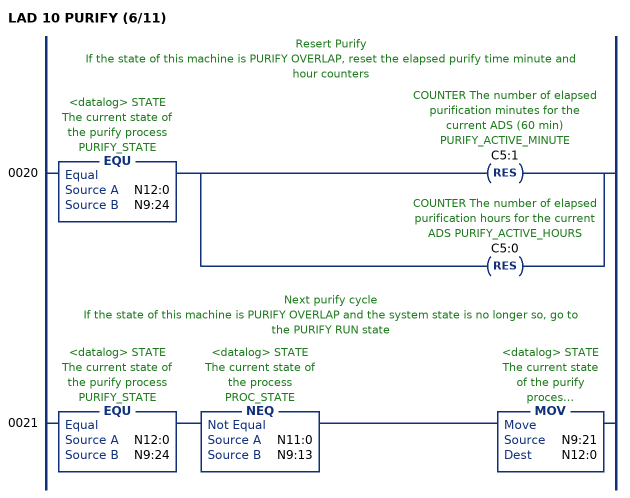
% Rung: 20 %
% Resert Purify
% If the state of this machine is PURIFY OVERLAP, reset the elapsed purify time minute and hour counters %
SOR EQU N12:0 N9:24 BST RES C5:1 NXB RES C5:0 BND EOR
%   N12:0  PURIFY_STATE  "<datalog> STATE The current state of the purify process" %
%   N9:24  PURIFY_OVERLAP  "STATE Puriify Overlap" %
%   C5:1  PURIFY_ACTIVE_MINUTE  "COUNTER The number of elapsed purification minutes for the current ADS (60 min)" %
%   C5:0  PURIFY_ACTIVE_HOURS  "COUNTER The number of elapsed purification hours for the current ADS" %
% Rung: 21 %
% Next purify cycle
% If the state of this machine is PURIFY OVERLAP and the system state is no longer so, go to the PURIFY RUN state %
SOR EQU N12:0 N9:24 NEQ N11:0 N9:13 MOV N9:21 N12:0 EOR
%   N12:0  PURIFY_STATE  "<datalog> STATE The current state of the purify process" %
%   N9:24  PURIFY_OVERLAP  "STATE Puriify Overlap" %
%   N11:0  PROC_STATE  "<datalog> STATE The current state of the process" %
%   N9:13  PROC_OVERLAP  "STATE Process Purify Overlap" %
%   N9:21  PURIFY_RUN  "STATE Purify running" %

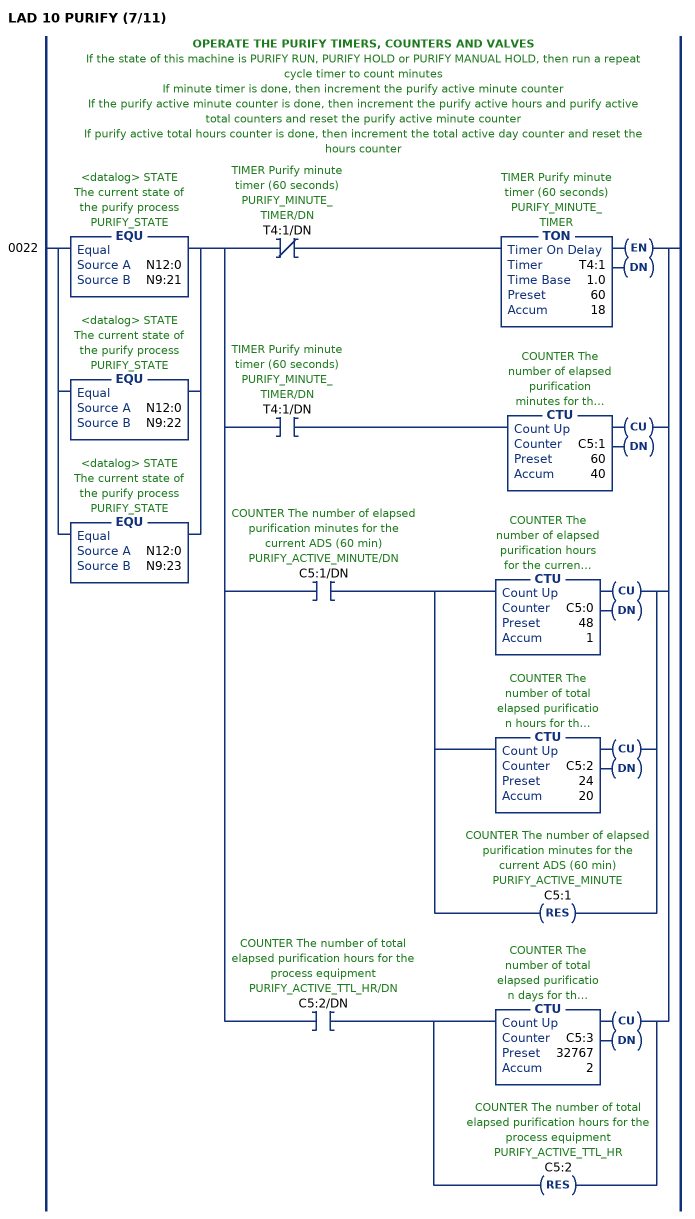
% Rung: 22 %
% TITLE: OPERATE THE PURIFY TIMERS, COUNTERS AND VALVES %
% If the state of this machine is PURIFY RUN, PURIFY HOLD or PURIFY MANUAL HOLD, then run a repeat cycle timer to count minutes
% If minute timer is done, then increment the purify active minute counter
% If the purify active minute counter is done, then increment the purify active hours and purify active total counters and reset the purify active minute counter
% If purify active total hours counter is done, then increment the total active day counter and reset the hours counter %
SOR BST EQU N12:0 N9:21 NXB EQU N12:0 N9:22 NXB EQU N12:0 N9:23 BND BST XIO T4:1/DN TON T4:1 1.0 60 18 NXB XIC T4:1/DN CTU C5:1 60 40 NXB XIC C5:1/DN BST CTU C5:0 48 1 NXB CTU C5:2 24 20 NXB RES C5:1 BND NXB XIC C5:2/DN BST CTU C5:3 32767 2 NXB RES C5:2 BND BND EOR
%   N12:0  PURIFY_STATE  "<datalog> STATE The current state of the purify process" %
%   N9:21  PURIFY_RUN  "STATE Purify running" %
%   N9:22  PURIFY_HOLD  "STATE Purify Hold" %
%   N9:23  PURIFY_MANUAL_HOLD  "STATE Purify Manual Hold" %
%   T4:1  PURIFY_MINUTE_TIMER  "TIMER Purify minute timer (60 seconds)" %
%   C5:1  PURIFY_ACTIVE_MINUTE  "COUNTER The number of elapsed purification minutes for the current ADS (60 min)" %
%   C5:0  PURIFY_ACTIVE_HOURS  "COUNTER The number of elapsed purification hours for the current ADS" %
%   C5:2  PURIFY_ACTIVE_TTL_HR  "COUNTER The number of total elapsed purification hours for the process equipment" %
%   C5:3  PURIFY_ACTIVE_TTL_DY  "COUNTER The number of total elapsed purification days for the process equipment" %

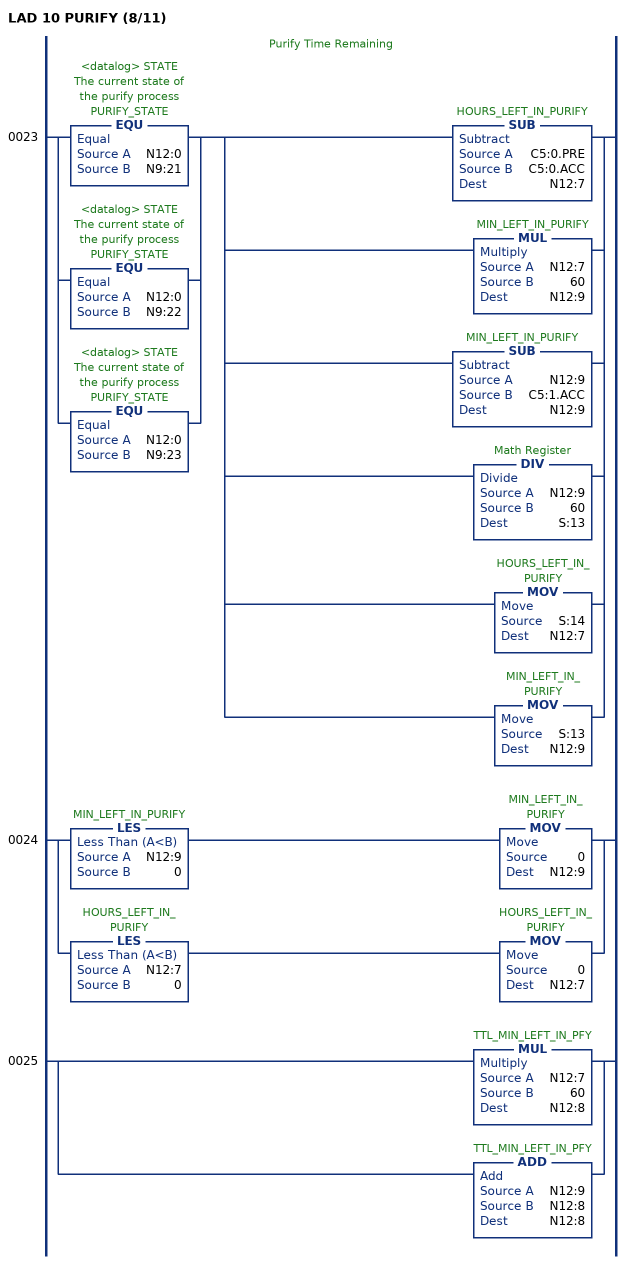
% Rung: 23 %
% Purify Time Remaining %
SOR BST EQU N12:0 N9:21 NXB EQU N12:0 N9:22 NXB EQU N12:0 N9:23 BND BST SUB C5:0.PRE C5:0.ACC N12:7 NXB MUL N12:7 60 N12:9 NXB SUB N12:9 C5:1.ACC N12:9 NXB DIV N12:9 60 S:13 NXB MOV S:14 N12:7 NXB MOV S:13 N12:9 BND EOR
%   N12:0  PURIFY_STATE  "<datalog> STATE The current state of the purify process" %
%   N9:21  PURIFY_RUN  "STATE Purify running" %
%   N9:22  PURIFY_HOLD  "STATE Purify Hold" %
%   N9:23  PURIFY_MANUAL_HOLD  "STATE Purify Manual Hold" %
%   C5:0  PURIFY_ACTIVE_HOURS  "COUNTER The number of elapsed purification hours for the current ADS" %
%   N12:7  HOURS_LEFT_IN_PURIFY %
%   N12:9  MIN_LEFT_IN_PURIFY %
%   C5:1  PURIFY_ACTIVE_MINUTE  "COUNTER The number of elapsed purification minutes for the current ADS (60 min)" %
%   S:13  "Math Register" %
%   S:14  "Math Register" %
% Rung: 24 %
SOR BST LES N12:9 0 MOV 0 N12:9 NXB LES N12:7 0 MOV 0 N12:7 BND EOR
%   N12:9  MIN_LEFT_IN_PURIFY %
%   N12:7  HOURS_LEFT_IN_PURIFY %
% Rung: 25 %
SOR BST MUL N12:7 60 N12:8 NXB ADD N12:9 N12:8 N12:8 BND EOR
%   N12:7  HOURS_LEFT_IN_PURIFY %
%   N12:8  TTL_MIN_LEFT_IN_PFY %
%   N12:9  MIN_LEFT_IN_PURIFY %

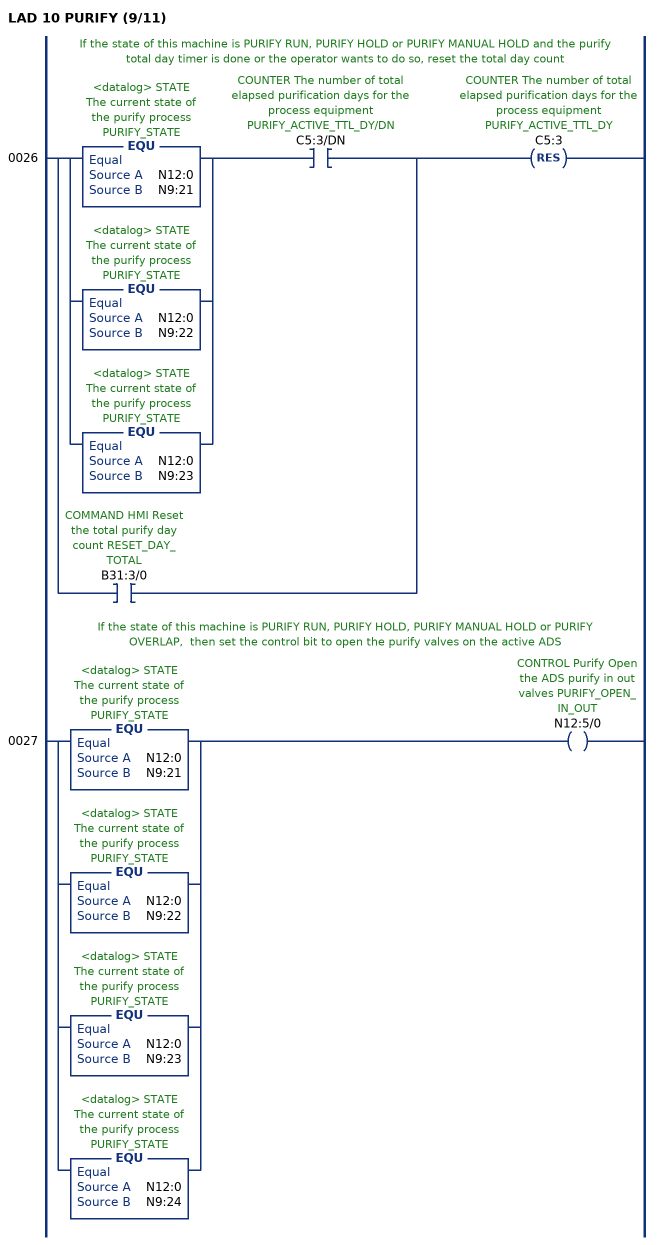
% Rung: 26 %
% If the state of this machine is PURIFY RUN, PURIFY HOLD or PURIFY MANUAL HOLD and the purify total day timer is done or the operator wants to do so, reset the total day count %
SOR BST BST EQU N12:0 N9:21 NXB EQU N12:0 N9:22 NXB EQU N12:0 N9:23 BND XIC C5:3/DN NXB XIC B31:3/0 BND RES C5:3 EOR
%   N12:0  PURIFY_STATE  "<datalog> STATE The current state of the purify process" %
%   N9:21  PURIFY_RUN  "STATE Purify running" %
%   N9:22  PURIFY_HOLD  "STATE Purify Hold" %
%   N9:23  PURIFY_MANUAL_HOLD  "STATE Purify Manual Hold" %
%   C5:3  PURIFY_ACTIVE_TTL_DY  "COUNTER The number of total elapsed purification days for the process equipment" %
%   B31:3/0  RESET_DAY_TOTAL  "COMMAND HMI Reset the total purify day count" %
% Rung: 27 %
% If the state of this machine is PURIFY RUN, PURIFY HOLD, PURIFY MANUAL HOLD or PURIFY OVERLAP,  then set the control bit to open the purify valves on the active ADS %
SOR BST EQU N12:0 N9:21 NXB EQU N12:0 N9:22 NXB EQU N12:0 N9:23 NXB EQU N12:0 N9:24 BND OTE N12:5/0 EOR
%   N12:0  PURIFY_STATE  "<datalog> STATE The current state of the purify process" %
%   N9:21  PURIFY_RUN  "STATE Purify running" %
%   N9:22  PURIFY_HOLD  "STATE Purify Hold" %
%   N9:23  PURIFY_MANUAL_HOLD  "STATE Purify Manual Hold" %
%   N9:24  PURIFY_OVERLAP  "STATE Puriify Overlap" %
%   N12:5/0  PURIFY_OPEN_IN_OUT  "CONTROL Purify Open the ADS purify in out valves" %

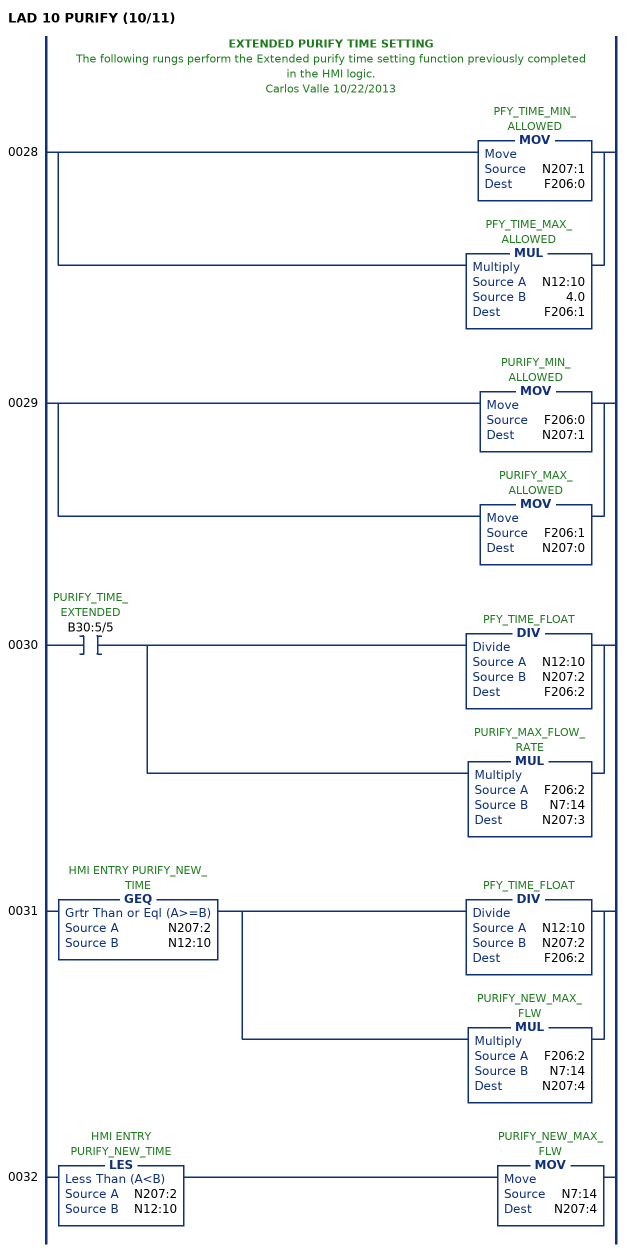
% Rung: 28 %
% TITLE: EXTENDED PURIFY TIME SETTING %
% The following rungs perform the Extended purify time setting function previously completed in the HMI logic.
% Carlos Valle 10/22/2013 %
SOR BST MOV N207:1 F206:0 NXB MUL N12:10 4.0 F206:1 BND EOR
%   N207:1  PURIFY_MIN_ALLOWED %
%   F206:0  PFY_TIME_MIN_ALLOWED %
%   N12:10  DEFAULT_PURIFY_TIME  "CONFIG The percent output requested by the operator (percent)" %
%   F206:1  PFY_TIME_MAX_ALLOWED %
% Rung: 29 %
SOR BST MOV F206:0 N207:1 NXB MOV F206:1 N207:0 BND EOR
%   F206:0  PFY_TIME_MIN_ALLOWED %
%   N207:1  PURIFY_MIN_ALLOWED %
%   F206:1  PFY_TIME_MAX_ALLOWED %
%   N207:0  PURIFY_MAX_ALLOWED %
% Rung: 30 %
SOR XIC B30:5/5 BST DIV N12:10 N207:2 F206:2 NXB MUL F206:2 N7:14 N207:3 BND EOR
%   B30:5/5  PURIFY_TIME_EXTENDED %
%   N12:10  DEFAULT_PURIFY_TIME  "CONFIG The percent output requested by the operator (percent)" %
%   N207:2  PURIFY_NEW_TIME  "HMI ENTRY" %
%   F206:2  PFY_TIME_FLOAT %
%   N7:14  PURIFIER_SIZE %
%   N207:3  PURIFY_MAX_FLOW_RATE %
% Rung: 31 %
SOR GEQ N207:2 N12:10 BST DIV N12:10 N207:2 F206:2 NXB MUL F206:2 N7:14 N207:4 BND EOR
%   N207:2  PURIFY_NEW_TIME  "HMI ENTRY" %
%   N12:10  DEFAULT_PURIFY_TIME  "CONFIG The percent output requested by the operator (percent)" %
%   F206:2  PFY_TIME_FLOAT %
%   N7:14  PURIFIER_SIZE %
%   N207:4  PURIFY_NEW_MAX_FLW %
% Rung: 32 %
SOR LES N207:2 N12:10 MOV N7:14 N207:4 EOR
%   N207:2  PURIFY_NEW_TIME  "HMI ENTRY" %
%   N12:10  DEFAULT_PURIFY_TIME  "CONFIG The percent output requested by the operator (percent)" %
%   N7:14  PURIFIER_SIZE %
%   N207:4  PURIFY_NEW_MAX_FLW %

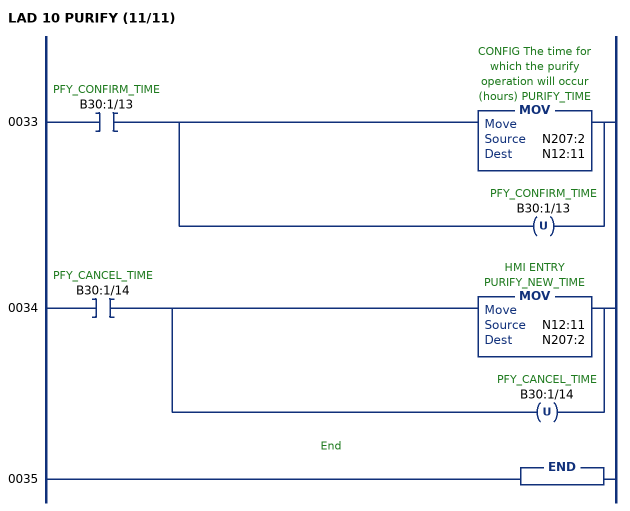
% Rung: 33 %
SOR XIC B30:1/13 BST MOV N207:2 N12:11 NXB OTU B30:1/13 BND EOR
%   B30:1/13  PFY_CONFIRM_TIME %
%   N207:2  PURIFY_NEW_TIME  "HMI ENTRY" %
%   N12:11  PURIFY_TIME  "CONFIG The time for which the purify operation will occur (hours)" %
% Rung: 34 %
SOR XIC B30:1/14 BST MOV N12:11 N207:2 NXB OTU B30:1/14 BND EOR
%   B30:1/14  PFY_CANCEL_TIME %
%   N12:11  PURIFY_TIME  "CONFIG The time for which the purify operation will occur (hours)" %
%   N207:2  PURIFY_NEW_TIME  "HMI ENTRY" %
% Rung: 35 %
% End %
SOR END EOR

LADDER 11 "REGEN"    % Operates the regen control %
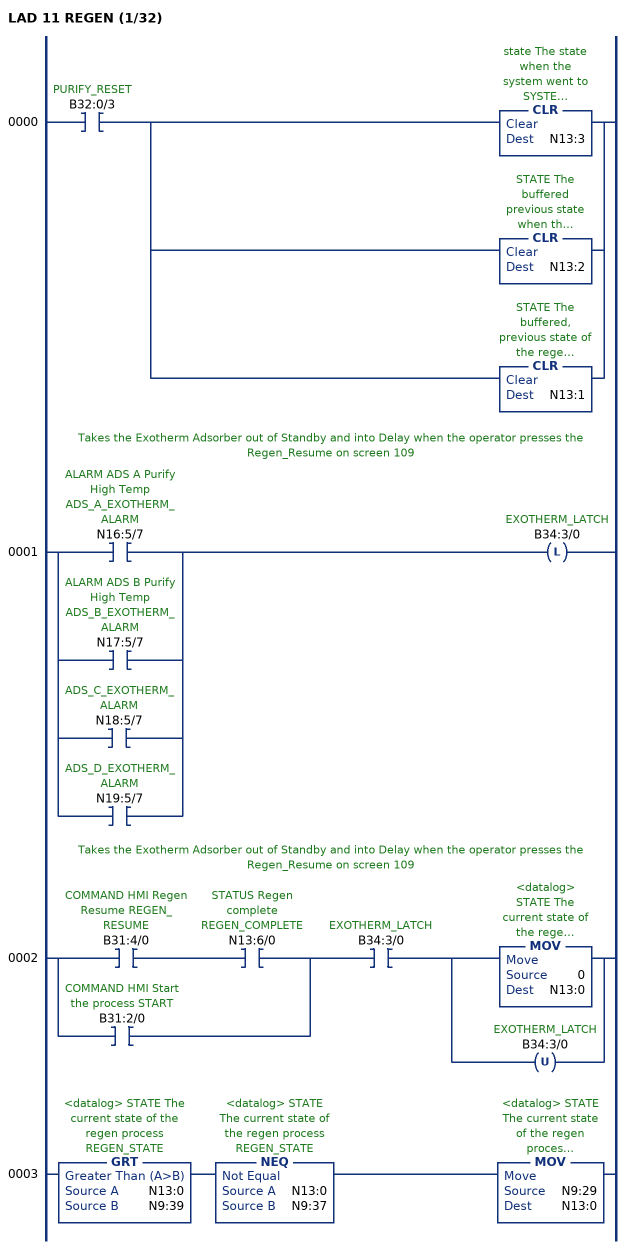
% Rung: 0 %
SOR XIC B32:0/3 BST CLR N13:3 NXB CLR N13:2 NXB CLR N13:1 BND EOR
%   B32:0/3  PURIFY_RESET %
%   N13:3  REGEN_STANDBY_BUFFER  "state The state when the system went to SYSTEM STANDBY" %
%   N13:2  REGEN_ALARM_BUFFER  "STATE The buffered previous state when the system alarm occured" %
%   N13:1  REGEN_BUFFER  "STATE The buffered, previous state of the regen process" %
% Rung: 1 %
% Takes the Exotherm Adsorber out of Standby and into Delay when the operator presses the Regen_Resume on screen 109 %
SOR BST XIC N16:5/7 NXB XIC N17:5/7 NXB XIC N18:5/7 NXB XIC N19:5/7 BND OTL B34:3/0 EOR
%   N16:5/7  ADS_A_EXOTHERM_ALARM  "ALARM ADS A Purify High Temp" %
%   N17:5/7  ADS_B_EXOTHERM_ALARM  "ALARM ADS B Purify High Temp" %
%   N18:5/7  ADS_C_EXOTHERM_ALARM %
%   N19:5/7  ADS_D_EXOTHERM_ALARM %
%   B34:3/0  EXOTHERM_LATCH %
% Rung: 2 %
% Takes the Exotherm Adsorber out of Standby and into Delay when the operator presses the Regen_Resume on screen 109 %
SOR BST XIC B31:4/0 XIC N13:6/0 NXB XIC B31:2/0 BND XIC B34:3/0 BST MOV 0 N13:0 NXB OTU B34:3/0 BND EOR
%   B31:4/0  REGEN_RESUME  "COMMAND HMI Regen Resume" %
%   N13:6/0  REGEN_COMPLETE  "STATUS Regen complete" %
%   B31:2/0  START  "COMMAND HMI Start the process" %
%   B34:3/0  EXOTHERM_LATCH %
%   N13:0  REGEN_STATE  "<datalog> STATE The current state of the regen process" %
% Rung: 3 %
SOR GRT N13:0 N9:39 NEQ N13:0 N9:37 MOV N9:29 N13:0 EOR
%   N13:0  REGEN_STATE  "<datalog> STATE The current state of the regen process" %
%   N9:39  REGEN_EQUALIZE  "STATE Regen Equalize" %
%   N9:37  REGEN_ALARM  "STATE Regen Alarm" %
%   N9:29  REGEN_IDLE  "STATE Regen Idle" %

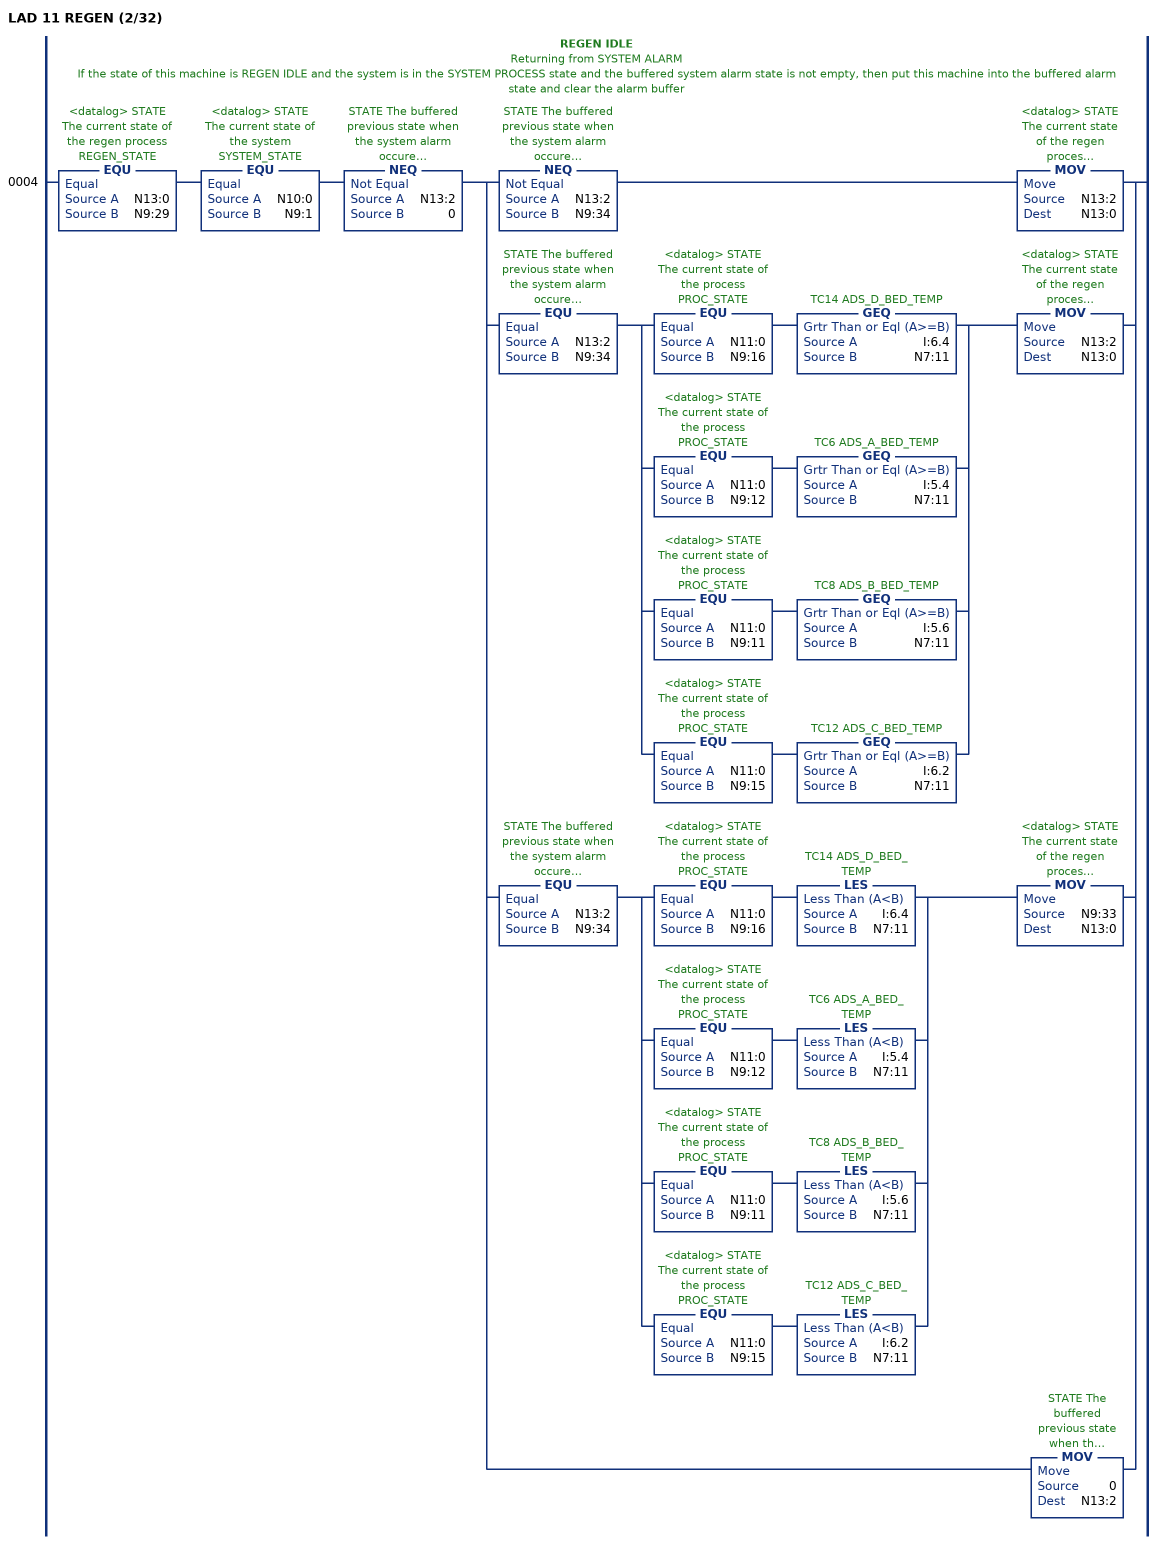
% Rung: 4 %
% TITLE: REGEN IDLE %
% Returning from SYSTEM ALARM
% If the state of this machine is REGEN IDLE and the system is in the SYSTEM PROCESS state and the buffered system alarm state is not empty, then put this machine into the buffered alarm state and clear the alarm buffer %
SOR EQU N13:0 N9:29 EQU N10:0 N9:1 NEQ N13:2 0 BST NEQ N13:2 N9:34 MOV N13:2 N13:0 NXB EQU N13:2 N9:34 BST EQU N11:0 N9:16 GEQ I:6.4 N7:11 NXB EQU N11:0 N9:12 GEQ I:5.4 N7:11 NXB EQU N11:0 N9:11 GEQ I:5.6 N7:11 NXB EQU N11:0 N9:15 GEQ I:6.2 N7:11 BND MOV N13:2 N13:0 NXB EQU N13:2 N9:34 BST EQU N11:0 N9:16 LES I:6.4 N7:11 NXB EQU N11:0 N9:12 LES I:5.4 N7:11 NXB EQU N11:0 N9:11 LES I:5.6 N7:11 NXB EQU N11:0 N9:15 LES I:6.2 N7:11 BND MOV N9:33 N13:0 NXB MOV 0 N13:2 BND EOR
%   N13:0  REGEN_STATE  "<datalog> STATE The current state of the regen process" %
%   N9:29  REGEN_IDLE  "STATE Regen Idle" %
%   N10:0  SYSTEM_STATE  "<datalog> STATE The current state of the system" %
%   N9:1  SYSTEM_PROCESS  "STATE System Process" %
%   N13:2  REGEN_ALARM_BUFFER  "STATE The buffered previous state when the system alarm occured" %
%   N9:34  REGEN_H2_REDUCTION  "STATE Regen Running" %
%   N11:0  PROC_STATE  "<datalog> STATE The current state of the process" %
%   N9:16  PROC_REGEN_D  "STATE Process Regen D" %
%   I:6.4  ADS_D_BED_TEMP  "TC14" %
%   N7:11  ADS_BED_TEMP_HIGH  "CONFIG The temp at which the regen process may continue" %
%   N9:12  PROC_REGEN_A  "STATE Process Regen A" %
%   I:5.4  ADS_A_BED_TEMP  "TC6" %
%   N9:11  PROC_REGEN_B  "STATE Process Regen B" %
%   I:5.6  ADS_B_BED_TEMP  "TC8" %
%   N9:15  PROC_REGEN_C  "STATE Process Regen C" %
%   I:6.2  ADS_C_BED_TEMP  "TC12" %
%   N9:33  REGEN_HEAT_BED  "STATE Regen Heat wall" %

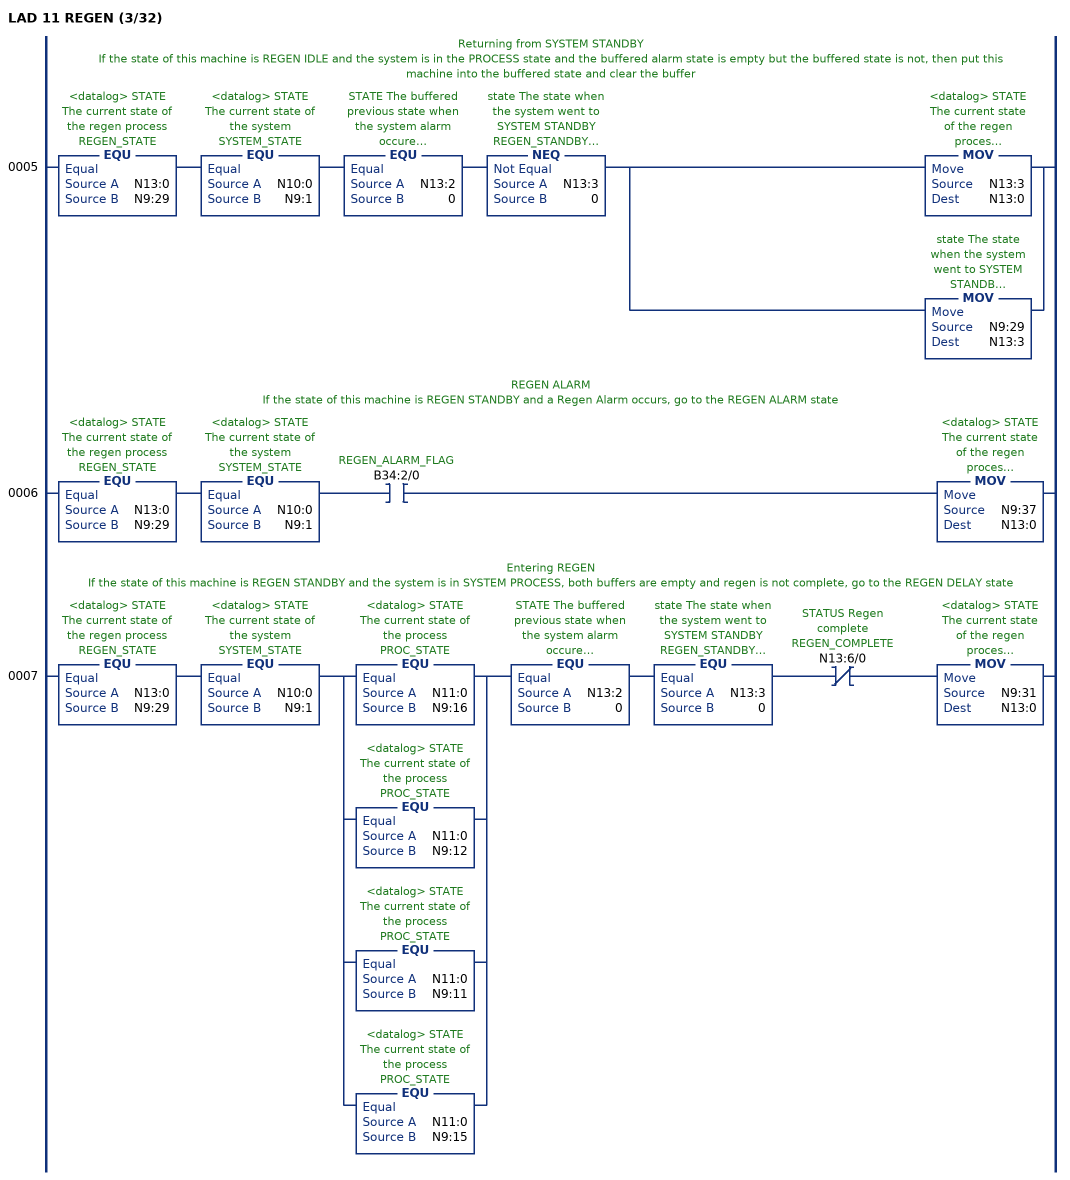
% Rung: 5 %
% Returning from SYSTEM STANDBY
% If the state of this machine is REGEN IDLE and the system is in the PROCESS state and the buffered alarm state is empty but the buffered state is not, then put this machine into the buffered state and clear the buffer %
SOR EQU N13:0 N9:29 EQU N10:0 N9:1 EQU N13:2 0 NEQ N13:3 0 BST MOV N13:3 N13:0 NXB MOV N9:29 N13:3 BND EOR
%   N13:0  REGEN_STATE  "<datalog> STATE The current state of the regen process" %
%   N9:29  REGEN_IDLE  "STATE Regen Idle" %
%   N10:0  SYSTEM_STATE  "<datalog> STATE The current state of the system" %
%   N9:1  SYSTEM_PROCESS  "STATE System Process" %
%   N13:2  REGEN_ALARM_BUFFER  "STATE The buffered previous state when the system alarm occured" %
%   N13:3  REGEN_STANDBY_BUFFER  "state The state when the system went to SYSTEM STANDBY" %
% Rung: 6 %
% REGEN ALARM
% If the state of this machine is REGEN STANDBY and a Regen Alarm occurs, go to the REGEN ALARM state %
SOR EQU N13:0 N9:29 EQU N10:0 N9:1 XIC B34:2/0 MOV N9:37 N13:0 EOR
%   N13:0  REGEN_STATE  "<datalog> STATE The current state of the regen process" %
%   N9:29  REGEN_IDLE  "STATE Regen Idle" %
%   N10:0  SYSTEM_STATE  "<datalog> STATE The current state of the system" %
%   N9:1  SYSTEM_PROCESS  "STATE System Process" %
%   B34:2/0  REGEN_ALARM_FLAG %
%   N9:37  REGEN_ALARM  "STATE Regen Alarm" %
% Rung: 7 %
% Entering REGEN
% If the state of this machine is REGEN STANDBY and the system is in SYSTEM PROCESS, both buffers are empty and regen is not complete, go to the REGEN DELAY state %
SOR EQU N13:0 N9:29 EQU N10:0 N9:1 BST EQU N11:0 N9:16 NXB EQU N11:0 N9:12 NXB EQU N11:0 N9:11 NXB EQU N11:0 N9:15 BND EQU N13:2 0 EQU N13:3 0 XIO N13:6/0 MOV N9:31 N13:0 EOR
%   N13:0  REGEN_STATE  "<datalog> STATE The current state of the regen process" %
%   N9:29  REGEN_IDLE  "STATE Regen Idle" %
%   N10:0  SYSTEM_STATE  "<datalog> STATE The current state of the system" %
%   N9:1  SYSTEM_PROCESS  "STATE System Process" %
%   N11:0  PROC_STATE  "<datalog> STATE The current state of the process" %
%   N9:16  PROC_REGEN_D  "STATE Process Regen D" %
%   N9:12  PROC_REGEN_A  "STATE Process Regen A" %
%   N9:11  PROC_REGEN_B  "STATE Process Regen B" %
%   N9:15  PROC_REGEN_C  "STATE Process Regen C" %
%   N13:2  REGEN_ALARM_BUFFER  "STATE The buffered previous state when the system alarm occured" %
%   N13:3  REGEN_STANDBY_BUFFER  "state The state when the system went to SYSTEM STANDBY" %
%   N13:6/0  REGEN_COMPLETE  "STATUS Regen complete" %
%   N9:31  REGEN_DELAY  "STATE Regen Delay" %

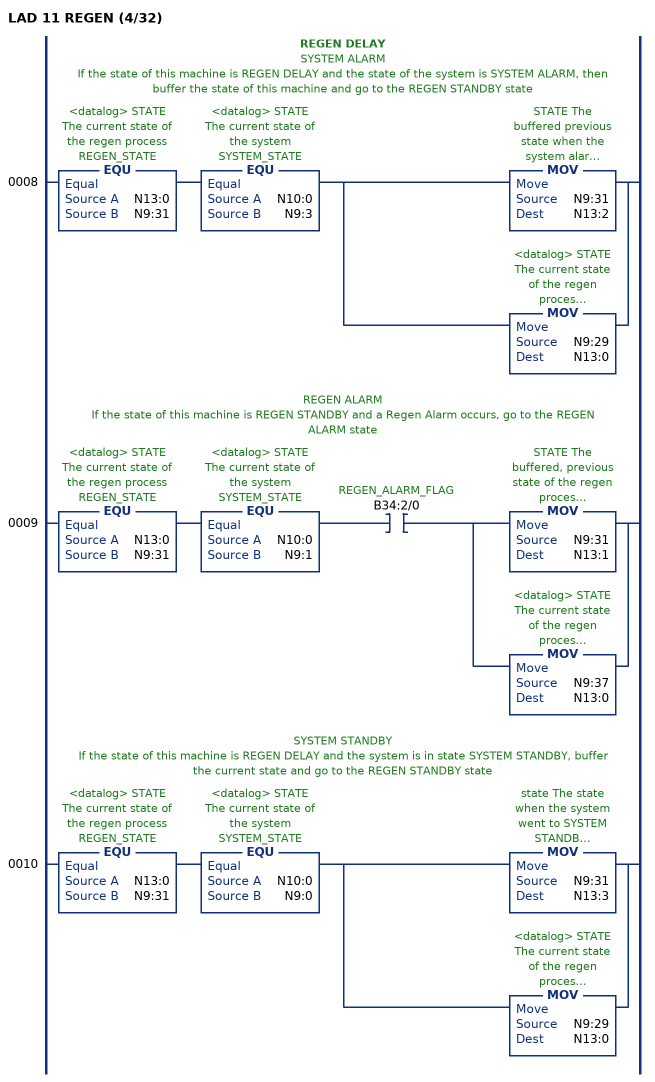
% Rung: 8 %
% TITLE: REGEN DELAY %
% SYSTEM ALARM
% If the state of this machine is REGEN DELAY and the state of the system is SYSTEM ALARM, then buffer the state of this machine and go to the REGEN STANDBY state %
SOR EQU N13:0 N9:31 EQU N10:0 N9:3 BST MOV N9:31 N13:2 NXB MOV N9:29 N13:0 BND EOR
%   N13:0  REGEN_STATE  "<datalog> STATE The current state of the regen process" %
%   N9:31  REGEN_DELAY  "STATE Regen Delay" %
%   N10:0  SYSTEM_STATE  "<datalog> STATE The current state of the system" %
%   N9:3  SYSTEM_ALARM  "STATE System Alarm" %
%   N13:2  REGEN_ALARM_BUFFER  "STATE The buffered previous state when the system alarm occured" %
%   N9:29  REGEN_IDLE  "STATE Regen Idle" %
% Rung: 9 %
% REGEN ALARM
% If the state of this machine is REGEN STANDBY and a Regen Alarm occurs, go to the REGEN ALARM state %
SOR EQU N13:0 N9:31 EQU N10:0 N9:1 XIC B34:2/0 BST MOV N9:31 N13:1 NXB MOV N9:37 N13:0 BND EOR
%   N13:0  REGEN_STATE  "<datalog> STATE The current state of the regen process" %
%   N9:31  REGEN_DELAY  "STATE Regen Delay" %
%   N10:0  SYSTEM_STATE  "<datalog> STATE The current state of the system" %
%   N9:1  SYSTEM_PROCESS  "STATE System Process" %
%   B34:2/0  REGEN_ALARM_FLAG %
%   N13:1  REGEN_BUFFER  "STATE The buffered, previous state of the regen process" %
%   N9:37  REGEN_ALARM  "STATE Regen Alarm" %
% Rung: 10 %
% SYSTEM STANDBY
% If the state of this machine is REGEN DELAY and the system is in state SYSTEM STANDBY, buffer the current state and go to the REGEN STANDBY state %
SOR EQU N13:0 N9:31 EQU N10:0 N9:0 BST MOV N9:31 N13:3 NXB MOV N9:29 N13:0 BND EOR
%   N13:0  REGEN_STATE  "<datalog> STATE The current state of the regen process" %
%   N9:31  REGEN_DELAY  "STATE Regen Delay" %
%   N10:0  SYSTEM_STATE  "<datalog> STATE The current state of the system" %
%   N9:0  SYSTEM_STANDBY  "STATE System Standby" %
%   N13:3  REGEN_STANDBY_BUFFER  "state The state when the system went to SYSTEM STANDBY" %
%   N9:29  REGEN_IDLE  "STATE Regen Idle" %

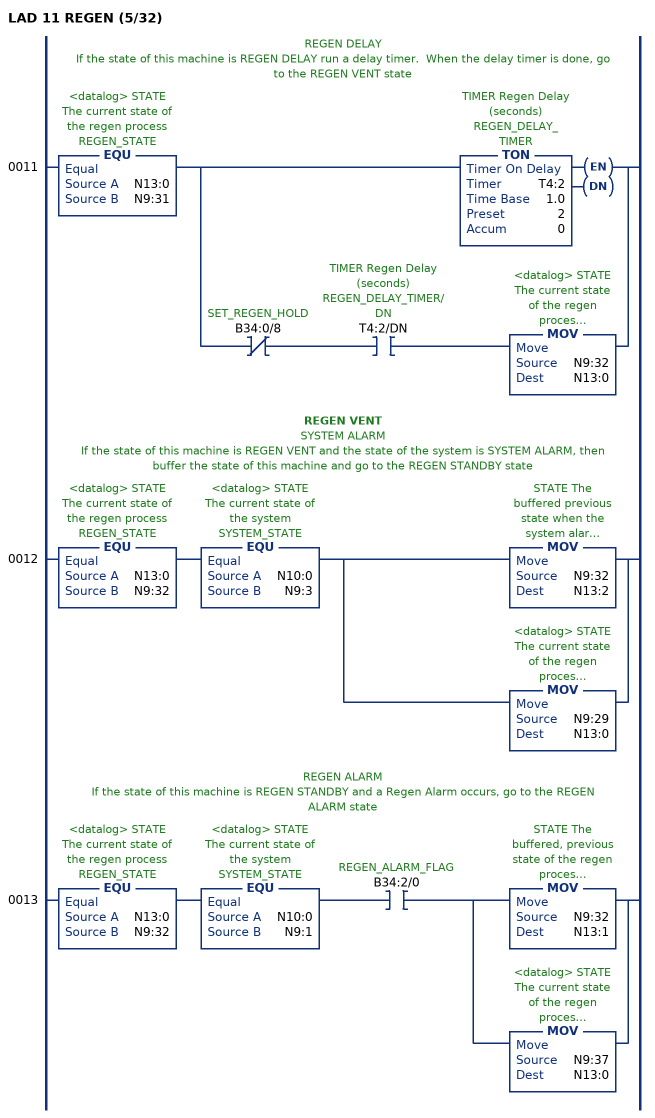
% Rung: 11 %
% REGEN DELAY
% If the state of this machine is REGEN DELAY run a delay timer.  When the delay timer is done, go to the REGEN VENT state %
SOR EQU N13:0 N9:31 BST TON T4:2 1.0 2 0 NXB XIO B34:0/8 XIC T4:2/DN MOV N9:32 N13:0 BND EOR
%   N13:0  REGEN_STATE  "<datalog> STATE The current state of the regen process" %
%   N9:31  REGEN_DELAY  "STATE Regen Delay" %
%   T4:2  REGEN_DELAY_TIMER  "TIMER Regen Delay (seconds)" %
%   B34:0/8  SET_REGEN_HOLD %
%   N9:32  REGEN_VENT  "STATE Regen Vent" %
% Rung: 12 %
% TITLE: REGEN VENT %
% SYSTEM ALARM
% If the state of this machine is REGEN VENT and the state of the system is SYSTEM ALARM, then buffer the state of this machine and go to the REGEN STANDBY state %
SOR EQU N13:0 N9:32 EQU N10:0 N9:3 BST MOV N9:32 N13:2 NXB MOV N9:29 N13:0 BND EOR
%   N13:0  REGEN_STATE  "<datalog> STATE The current state of the regen process" %
%   N9:32  REGEN_VENT  "STATE Regen Vent" %
%   N10:0  SYSTEM_STATE  "<datalog> STATE The current state of the system" %
%   N9:3  SYSTEM_ALARM  "STATE System Alarm" %
%   N13:2  REGEN_ALARM_BUFFER  "STATE The buffered previous state when the system alarm occured" %
%   N9:29  REGEN_IDLE  "STATE Regen Idle" %
% Rung: 13 %
% REGEN ALARM
% If the state of this machine is REGEN STANDBY and a Regen Alarm occurs, go to the REGEN ALARM state %
SOR EQU N13:0 N9:32 EQU N10:0 N9:1 XIC B34:2/0 BST MOV N9:32 N13:1 NXB MOV N9:37 N13:0 BND EOR
%   N13:0  REGEN_STATE  "<datalog> STATE The current state of the regen process" %
%   N9:32  REGEN_VENT  "STATE Regen Vent" %
%   N10:0  SYSTEM_STATE  "<datalog> STATE The current state of the system" %
%   N9:1  SYSTEM_PROCESS  "STATE System Process" %
%   B34:2/0  REGEN_ALARM_FLAG %
%   N13:1  REGEN_BUFFER  "STATE The buffered, previous state of the regen process" %
%   N9:37  REGEN_ALARM  "STATE Regen Alarm" %

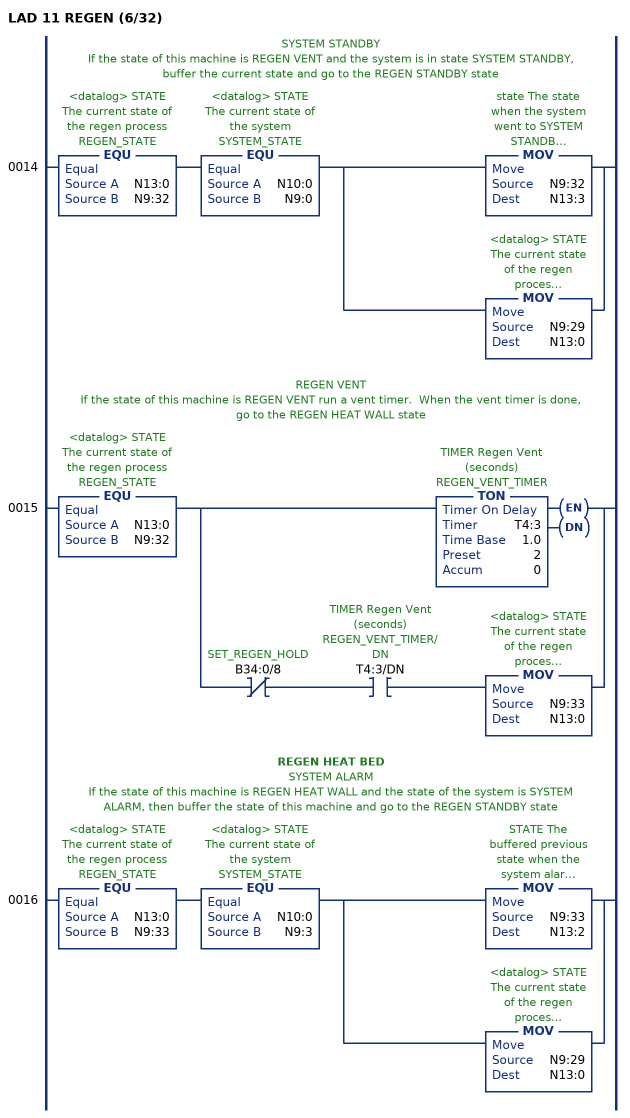
% Rung: 14 %
% SYSTEM STANDBY
% If the state of this machine is REGEN VENT and the system is in state SYSTEM STANDBY, buffer the current state and go to the REGEN STANDBY state %
SOR EQU N13:0 N9:32 EQU N10:0 N9:0 BST MOV N9:32 N13:3 NXB MOV N9:29 N13:0 BND EOR
%   N13:0  REGEN_STATE  "<datalog> STATE The current state of the regen process" %
%   N9:32  REGEN_VENT  "STATE Regen Vent" %
%   N10:0  SYSTEM_STATE  "<datalog> STATE The current state of the system" %
%   N9:0  SYSTEM_STANDBY  "STATE System Standby" %
%   N13:3  REGEN_STANDBY_BUFFER  "state The state when the system went to SYSTEM STANDBY" %
%   N9:29  REGEN_IDLE  "STATE Regen Idle" %
% Rung: 15 %
% REGEN VENT
% If the state of this machine is REGEN VENT run a vent timer.  When the vent timer is done, go to the REGEN HEAT WALL state %
SOR EQU N13:0 N9:32 BST TON T4:3 1.0 2 0 NXB XIO B34:0/8 XIC T4:3/DN MOV N9:33 N13:0 BND EOR
%   N13:0  REGEN_STATE  "<datalog> STATE The current state of the regen process" %
%   N9:32  REGEN_VENT  "STATE Regen Vent" %
%   T4:3  REGEN_VENT_TIMER  "TIMER Regen Vent (seconds)" %
%   B34:0/8  SET_REGEN_HOLD %
%   N9:33  REGEN_HEAT_BED  "STATE Regen Heat wall" %
% Rung: 16 %
% TITLE: REGEN HEAT BED %
% SYSTEM ALARM
% If the state of this machine is REGEN HEAT WALL and the state of the system is SYSTEM ALARM, then buffer the state of this machine and go to the REGEN STANDBY state %
SOR EQU N13:0 N9:33 EQU N10:0 N9:3 BST MOV N9:33 N13:2 NXB MOV N9:29 N13:0 BND EOR
%   N13:0  REGEN_STATE  "<datalog> STATE The current state of the regen process" %
%   N9:33  REGEN_HEAT_BED  "STATE Regen Heat wall" %
%   N10:0  SYSTEM_STATE  "<datalog> STATE The current state of the system" %
%   N9:3  SYSTEM_ALARM  "STATE System Alarm" %
%   N13:2  REGEN_ALARM_BUFFER  "STATE The buffered previous state when the system alarm occured" %
%   N9:29  REGEN_IDLE  "STATE Regen Idle" %

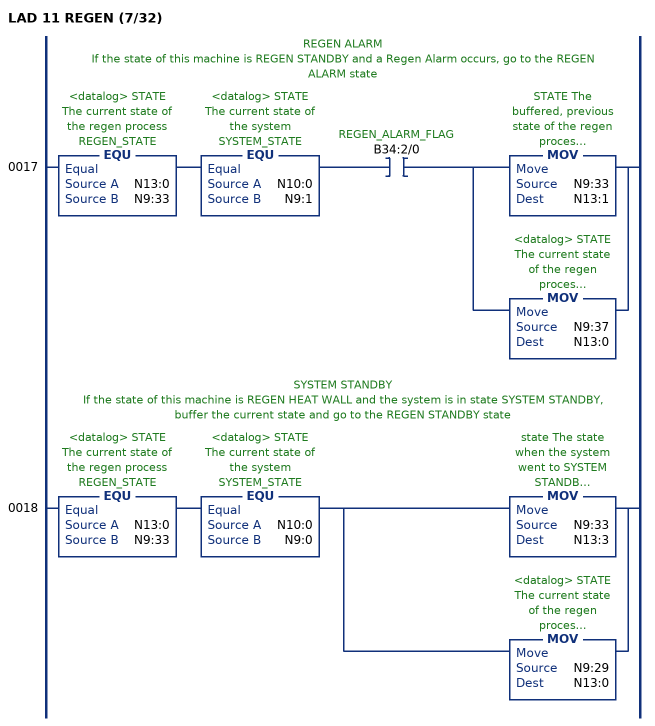
% Rung: 17 %
% REGEN ALARM
% If the state of this machine is REGEN STANDBY and a Regen Alarm occurs, go to the REGEN ALARM state %
SOR EQU N13:0 N9:33 EQU N10:0 N9:1 XIC B34:2/0 BST MOV N9:33 N13:1 NXB MOV N9:37 N13:0 BND EOR
%   N13:0  REGEN_STATE  "<datalog> STATE The current state of the regen process" %
%   N9:33  REGEN_HEAT_BED  "STATE Regen Heat wall" %
%   N10:0  SYSTEM_STATE  "<datalog> STATE The current state of the system" %
%   N9:1  SYSTEM_PROCESS  "STATE System Process" %
%   B34:2/0  REGEN_ALARM_FLAG %
%   N13:1  REGEN_BUFFER  "STATE The buffered, previous state of the regen process" %
%   N9:37  REGEN_ALARM  "STATE Regen Alarm" %
% Rung: 18 %
% SYSTEM STANDBY
% If the state of this machine is REGEN HEAT WALL and the system is in state SYSTEM STANDBY, buffer the current state and go to the REGEN STANDBY state %
SOR EQU N13:0 N9:33 EQU N10:0 N9:0 BST MOV N9:33 N13:3 NXB MOV N9:29 N13:0 BND EOR
%   N13:0  REGEN_STATE  "<datalog> STATE The current state of the regen process" %
%   N9:33  REGEN_HEAT_BED  "STATE Regen Heat wall" %
%   N10:0  SYSTEM_STATE  "<datalog> STATE The current state of the system" %
%   N9:0  SYSTEM_STANDBY  "STATE System Standby" %
%   N13:3  REGEN_STANDBY_BUFFER  "state The state when the system went to SYSTEM STANDBY" %
%   N9:29  REGEN_IDLE  "STATE Regen Idle" %

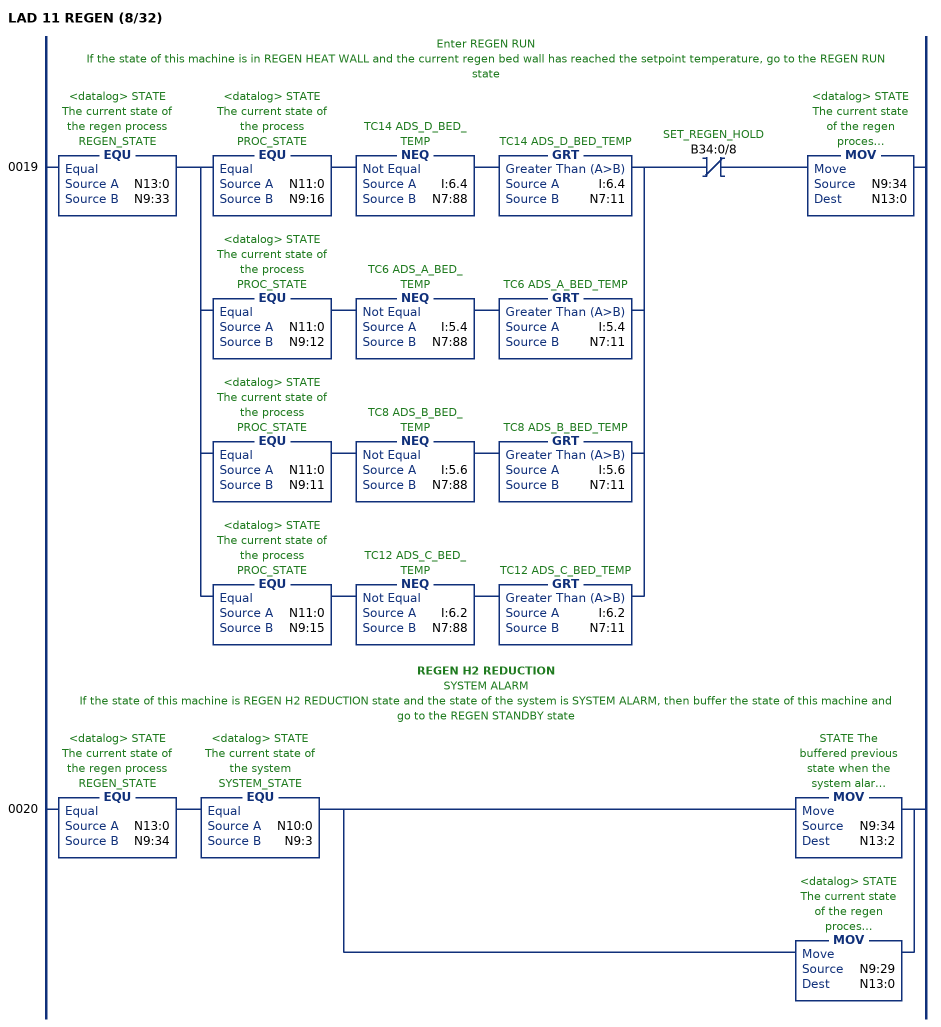
% Rung: 19 %
% Enter REGEN RUN
% If the state of this machine is in REGEN HEAT WALL and the current regen bed wall has reached the setpoint temperature, go to the REGEN RUN state %
SOR EQU N13:0 N9:33 BST EQU N11:0 N9:16 NEQ I:6.4 N7:88 GRT I:6.4 N7:11 NXB EQU N11:0 N9:12 NEQ I:5.4 N7:88 GRT I:5.4 N7:11 NXB EQU N11:0 N9:11 NEQ I:5.6 N7:88 GRT I:5.6 N7:11 NXB EQU N11:0 N9:15 NEQ I:6.2 N7:88 GRT I:6.2 N7:11 BND XIO B34:0/8 MOV N9:34 N13:0 EOR
%   N13:0  REGEN_STATE  "<datalog> STATE The current state of the regen process" %
%   N9:33  REGEN_HEAT_BED  "STATE Regen Heat wall" %
%   N11:0  PROC_STATE  "<datalog> STATE The current state of the process" %
%   N9:16  PROC_REGEN_D  "STATE Process Regen D" %
%   I:6.4  ADS_D_BED_TEMP  "TC14" %
%   N7:88  TC_OPEN_SP  "CONFIG TC Open Setpoint" %
%   N7:11  ADS_BED_TEMP_HIGH  "CONFIG The temp at which the regen process may continue" %
%   N9:12  PROC_REGEN_A  "STATE Process Regen A" %
%   I:5.4  ADS_A_BED_TEMP  "TC6" %
%   N9:11  PROC_REGEN_B  "STATE Process Regen B" %
%   I:5.6  ADS_B_BED_TEMP  "TC8" %
%   N9:15  PROC_REGEN_C  "STATE Process Regen C" %
%   I:6.2  ADS_C_BED_TEMP  "TC12" %
%   B34:0/8  SET_REGEN_HOLD %
%   N9:34  REGEN_H2_REDUCTION  "STATE Regen Running" %
% Rung: 20 %
% TITLE: REGEN H2 REDUCTION %
% SYSTEM ALARM
% If the state of this machine is REGEN H2 REDUCTION state and the state of the system is SYSTEM ALARM, then buffer the state of this machine and go to the REGEN STANDBY state %
SOR EQU N13:0 N9:34 EQU N10:0 N9:3 BST MOV N9:34 N13:2 NXB MOV N9:29 N13:0 BND EOR
%   N13:0  REGEN_STATE  "<datalog> STATE The current state of the regen process" %
%   N9:34  REGEN_H2_REDUCTION  "STATE Regen Running" %
%   N10:0  SYSTEM_STATE  "<datalog> STATE The current state of the system" %
%   N9:3  SYSTEM_ALARM  "STATE System Alarm" %
%   N13:2  REGEN_ALARM_BUFFER  "STATE The buffered previous state when the system alarm occured" %
%   N9:29  REGEN_IDLE  "STATE Regen Idle" %

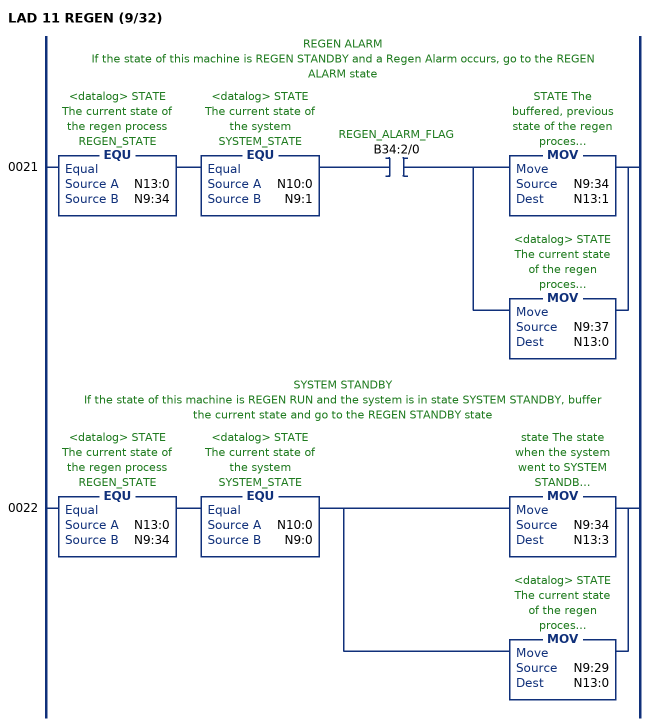
% Rung: 21 %
% REGEN ALARM
% If the state of this machine is REGEN STANDBY and a Regen Alarm occurs, go to the REGEN ALARM state %
SOR EQU N13:0 N9:34 EQU N10:0 N9:1 XIC B34:2/0 BST MOV N9:34 N13:1 NXB MOV N9:37 N13:0 BND EOR
%   N13:0  REGEN_STATE  "<datalog> STATE The current state of the regen process" %
%   N9:34  REGEN_H2_REDUCTION  "STATE Regen Running" %
%   N10:0  SYSTEM_STATE  "<datalog> STATE The current state of the system" %
%   N9:1  SYSTEM_PROCESS  "STATE System Process" %
%   B34:2/0  REGEN_ALARM_FLAG %
%   N13:1  REGEN_BUFFER  "STATE The buffered, previous state of the regen process" %
%   N9:37  REGEN_ALARM  "STATE Regen Alarm" %
% Rung: 22 %
% SYSTEM STANDBY
% If the state of this machine is REGEN RUN and the system is in state SYSTEM STANDBY, buffer the current state and go to the REGEN STANDBY state %
SOR EQU N13:0 N9:34 EQU N10:0 N9:0 BST MOV N9:34 N13:3 NXB MOV N9:29 N13:0 BND EOR
%   N13:0  REGEN_STATE  "<datalog> STATE The current state of the regen process" %
%   N9:34  REGEN_H2_REDUCTION  "STATE Regen Running" %
%   N10:0  SYSTEM_STATE  "<datalog> STATE The current state of the system" %
%   N9:0  SYSTEM_STANDBY  "STATE System Standby" %
%   N13:3  REGEN_STANDBY_BUFFER  "state The state when the system went to SYSTEM STANDBY" %
%   N9:29  REGEN_IDLE  "STATE Regen Idle" %

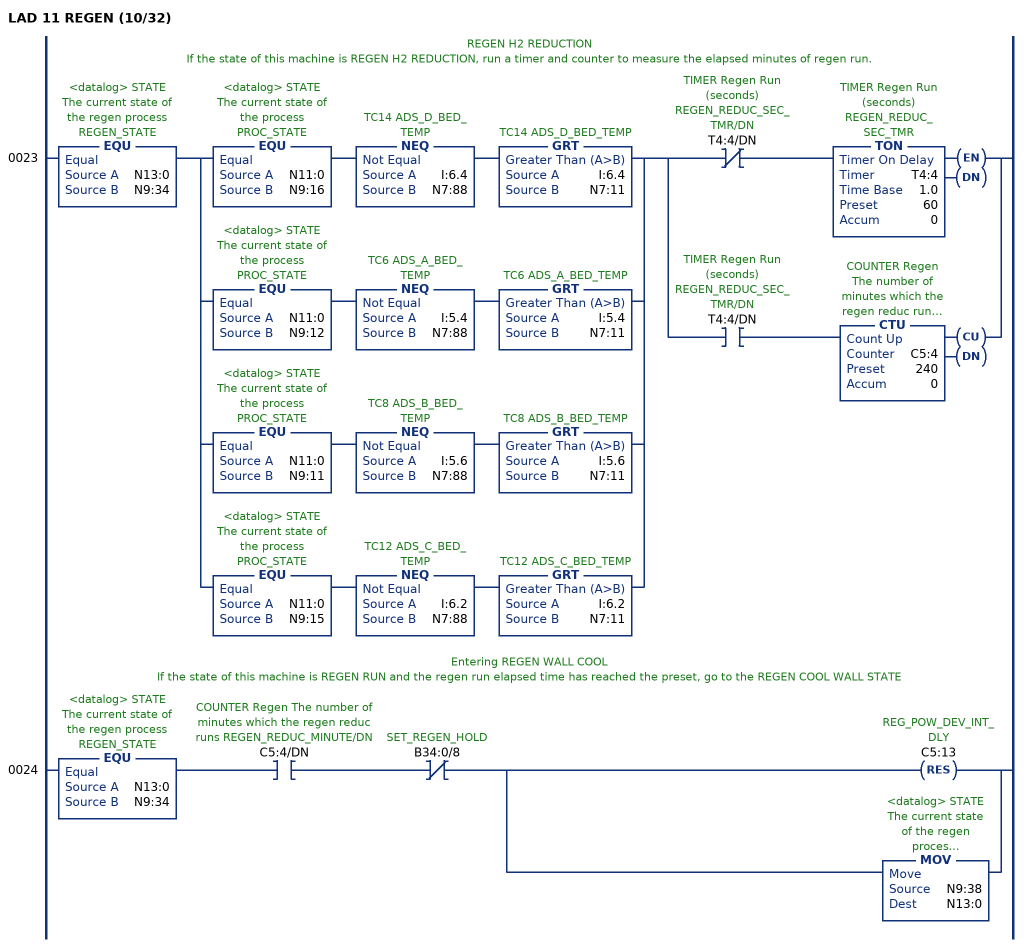
% Rung: 23 %
% REGEN H2 REDUCTION
% If the state of this machine is REGEN H2 REDUCTION, run a timer and counter to measure the elapsed minutes of regen run. %
SOR EQU N13:0 N9:34 BST EQU N11:0 N9:16 NEQ I:6.4 N7:88 GRT I:6.4 N7:11 NXB EQU N11:0 N9:12 NEQ I:5.4 N7:88 GRT I:5.4 N7:11 NXB EQU N11:0 N9:11 NEQ I:5.6 N7:88 GRT I:5.6 N7:11 NXB EQU N11:0 N9:15 NEQ I:6.2 N7:88 GRT I:6.2 N7:11 BND BST XIO T4:4/DN TON T4:4 1.0 60 0 NXB XIC T4:4/DN CTU C5:4 240 0 BND EOR
%   N13:0  REGEN_STATE  "<datalog> STATE The current state of the regen process" %
%   N9:34  REGEN_H2_REDUCTION  "STATE Regen Running" %
%   N11:0  PROC_STATE  "<datalog> STATE The current state of the process" %
%   N9:16  PROC_REGEN_D  "STATE Process Regen D" %
%   I:6.4  ADS_D_BED_TEMP  "TC14" %
%   N7:88  TC_OPEN_SP  "CONFIG TC Open Setpoint" %
%   N7:11  ADS_BED_TEMP_HIGH  "CONFIG The temp at which the regen process may continue" %
%   N9:12  PROC_REGEN_A  "STATE Process Regen A" %
%   I:5.4  ADS_A_BED_TEMP  "TC6" %
%   N9:11  PROC_REGEN_B  "STATE Process Regen B" %
%   I:5.6  ADS_B_BED_TEMP  "TC8" %
%   N9:15  PROC_REGEN_C  "STATE Process Regen C" %
%   I:6.2  ADS_C_BED_TEMP  "TC12" %
%   T4:4  REGEN_REDUC_SEC_TMR  "TIMER Regen Run (seconds)" %
%   C5:4  REGEN_REDUC_MINUTE  "COUNTER Regen The number of minutes which the regen reduc runs" %
% Rung: 24 %
% Entering REGEN WALL COOL
% If the state of this machine is REGEN RUN and the regen run elapsed time has reached the preset, go to the REGEN COOL WALL STATE %
SOR EQU N13:0 N9:34 XIC C5:4/DN XIO B34:0/8 BST RES C5:13 NXB MOV N9:38 N13:0 BND EOR
%   N13:0  REGEN_STATE  "<datalog> STATE The current state of the regen process" %
%   N9:34  REGEN_H2_REDUCTION  "STATE Regen Running" %
%   C5:4  REGEN_REDUC_MINUTE  "COUNTER Regen The number of minutes which the regen reduc runs" %
%   B34:0/8  SET_REGEN_HOLD %
%   C5:13  REG_POW_DEV_INT_DLY %
%   N9:38  REGEN_PURGE  "STATE Regen Hot Purge" %

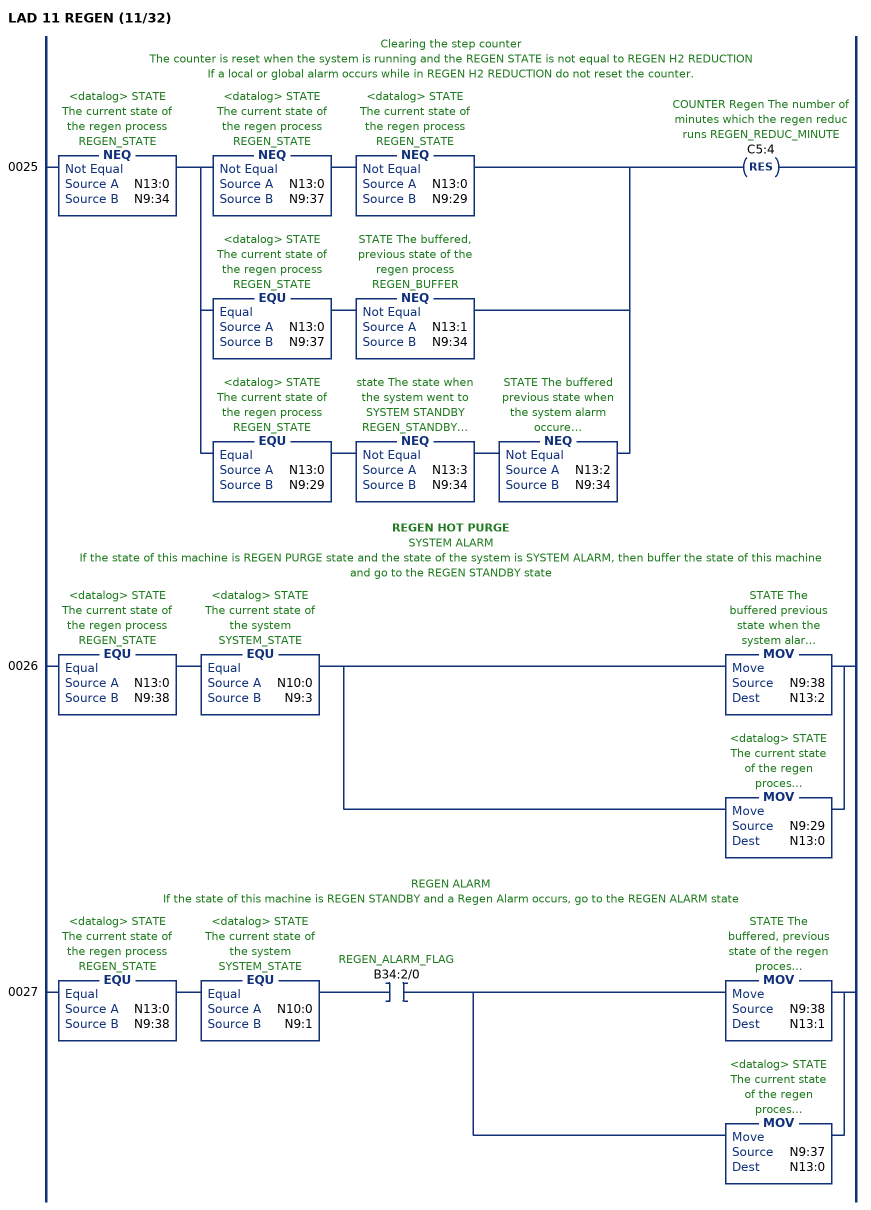
% Rung: 25 %
% Clearing the step counter
% The counter is reset when the system is running and the REGEN STATE is not equal to REGEN H2 REDUCTION
% If a local or global alarm occurs while in REGEN H2 REDUCTION do not reset the counter. %
SOR NEQ N13:0 N9:34 BST NEQ N13:0 N9:37 NEQ N13:0 N9:29 NXB EQU N13:0 N9:37 NEQ N13:1 N9:34 NXB EQU N13:0 N9:29 NEQ N13:3 N9:34 NEQ N13:2 N9:34 BND RES C5:4 EOR
%   N13:0  REGEN_STATE  "<datalog> STATE The current state of the regen process" %
%   N9:34  REGEN_H2_REDUCTION  "STATE Regen Running" %
%   N9:37  REGEN_ALARM  "STATE Regen Alarm" %
%   N9:29  REGEN_IDLE  "STATE Regen Idle" %
%   N13:1  REGEN_BUFFER  "STATE The buffered, previous state of the regen process" %
%   N13:3  REGEN_STANDBY_BUFFER  "state The state when the system went to SYSTEM STANDBY" %
%   N13:2  REGEN_ALARM_BUFFER  "STATE The buffered previous state when the system alarm occured" %
%   C5:4  REGEN_REDUC_MINUTE  "COUNTER Regen The number of minutes which the regen reduc runs" %
% Rung: 26 %
% TITLE: REGEN HOT PURGE %
% SYSTEM ALARM
% If the state of this machine is REGEN PURGE state and the state of the system is SYSTEM ALARM, then buffer the state of this machine and go to the REGEN STANDBY state %
SOR EQU N13:0 N9:38 EQU N10:0 N9:3 BST MOV N9:38 N13:2 NXB MOV N9:29 N13:0 BND EOR
%   N13:0  REGEN_STATE  "<datalog> STATE The current state of the regen process" %
%   N9:38  REGEN_PURGE  "STATE Regen Hot Purge" %
%   N10:0  SYSTEM_STATE  "<datalog> STATE The current state of the system" %
%   N9:3  SYSTEM_ALARM  "STATE System Alarm" %
%   N13:2  REGEN_ALARM_BUFFER  "STATE The buffered previous state when the system alarm occured" %
%   N9:29  REGEN_IDLE  "STATE Regen Idle" %
% Rung: 27 %
% REGEN ALARM
% If the state of this machine is REGEN STANDBY and a Regen Alarm occurs, go to the REGEN ALARM state %
SOR EQU N13:0 N9:38 EQU N10:0 N9:1 XIC B34:2/0 BST MOV N9:38 N13:1 NXB MOV N9:37 N13:0 BND EOR
%   N13:0  REGEN_STATE  "<datalog> STATE The current state of the regen process" %
%   N9:38  REGEN_PURGE  "STATE Regen Hot Purge" %
%   N10:0  SYSTEM_STATE  "<datalog> STATE The current state of the system" %
%   N9:1  SYSTEM_PROCESS  "STATE System Process" %
%   B34:2/0  REGEN_ALARM_FLAG %
%   N13:1  REGEN_BUFFER  "STATE The buffered, previous state of the regen process" %
%   N9:37  REGEN_ALARM  "STATE Regen Alarm" %

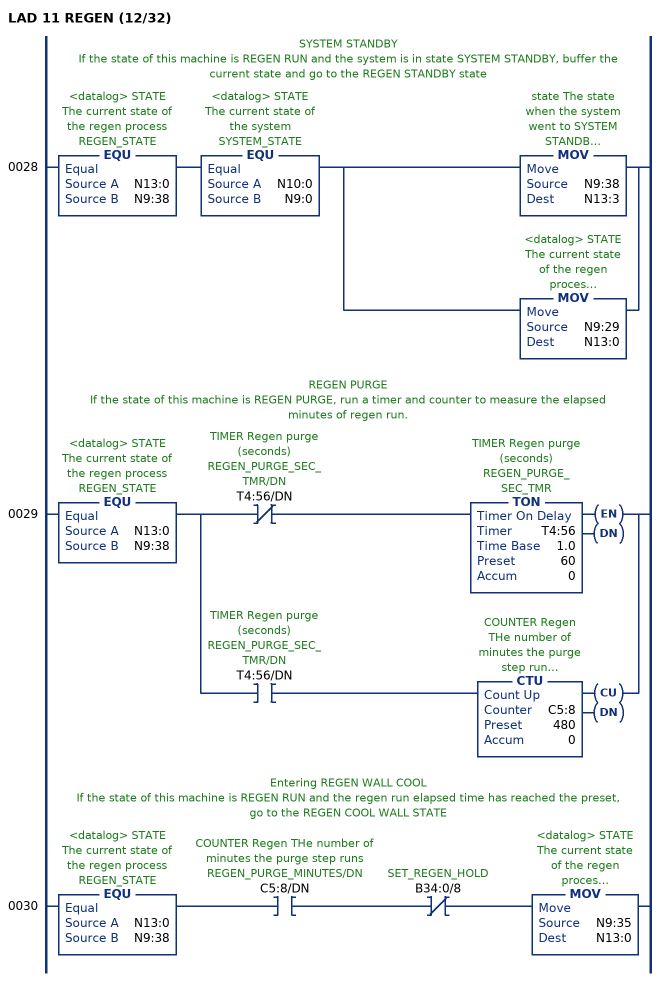
% Rung: 28 %
% SYSTEM STANDBY
% If the state of this machine is REGEN RUN and the system is in state SYSTEM STANDBY, buffer the current state and go to the REGEN STANDBY state %
SOR EQU N13:0 N9:38 EQU N10:0 N9:0 BST MOV N9:38 N13:3 NXB MOV N9:29 N13:0 BND EOR
%   N13:0  REGEN_STATE  "<datalog> STATE The current state of the regen process" %
%   N9:38  REGEN_PURGE  "STATE Regen Hot Purge" %
%   N10:0  SYSTEM_STATE  "<datalog> STATE The current state of the system" %
%   N9:0  SYSTEM_STANDBY  "STATE System Standby" %
%   N13:3  REGEN_STANDBY_BUFFER  "state The state when the system went to SYSTEM STANDBY" %
%   N9:29  REGEN_IDLE  "STATE Regen Idle" %
% Rung: 29 %
% REGEN PURGE
% If the state of this machine is REGEN PURGE, run a timer and counter to measure the elapsed minutes of regen run. %
SOR EQU N13:0 N9:38 BST XIO T4:56/DN TON T4:56 1.0 60 0 NXB XIC T4:56/DN CTU C5:8 480 0 BND EOR
%   N13:0  REGEN_STATE  "<datalog> STATE The current state of the regen process" %
%   N9:38  REGEN_PURGE  "STATE Regen Hot Purge" %
%   T4:56  REGEN_PURGE_SEC_TMR  "TIMER Regen purge (seconds)" %
%   C5:8  REGEN_PURGE_MINUTES  "COUNTER Regen THe number of minutes the purge step runs" %
% Rung: 30 %
% Entering REGEN WALL COOL
% If the state of this machine is REGEN RUN and the regen run elapsed time has reached the preset, go to the REGEN COOL WALL STATE %
SOR EQU N13:0 N9:38 XIC C5:8/DN XIO B34:0/8 MOV N9:35 N13:0 EOR
%   N13:0  REGEN_STATE  "<datalog> STATE The current state of the regen process" %
%   N9:38  REGEN_PURGE  "STATE Regen Hot Purge" %
%   C5:8  REGEN_PURGE_MINUTES  "COUNTER Regen THe number of minutes the purge step runs" %
%   B34:0/8  SET_REGEN_HOLD %
%   N9:35  REGEN_COOL_WALL  "STATE Regen Cool wall" %

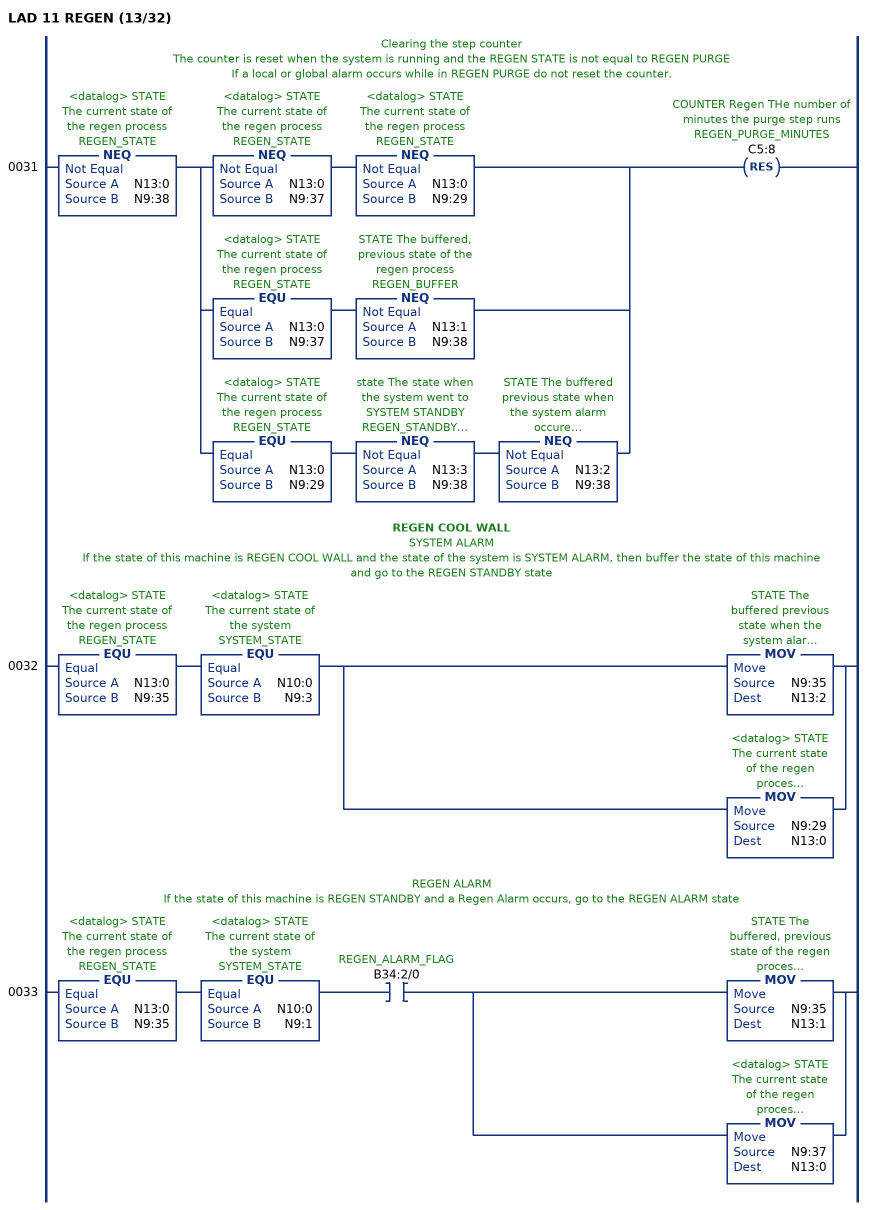
% Rung: 31 %
% Clearing the step counter
% The counter is reset when the system is running and the REGEN STATE is not equal to REGEN PURGE
% If a local or global alarm occurs while in REGEN PURGE do not reset the counter. %
SOR NEQ N13:0 N9:38 BST NEQ N13:0 N9:37 NEQ N13:0 N9:29 NXB EQU N13:0 N9:37 NEQ N13:1 N9:38 NXB EQU N13:0 N9:29 NEQ N13:3 N9:38 NEQ N13:2 N9:38 BND RES C5:8 EOR
%   N13:0  REGEN_STATE  "<datalog> STATE The current state of the regen process" %
%   N9:38  REGEN_PURGE  "STATE Regen Hot Purge" %
%   N9:37  REGEN_ALARM  "STATE Regen Alarm" %
%   N9:29  REGEN_IDLE  "STATE Regen Idle" %
%   N13:1  REGEN_BUFFER  "STATE The buffered, previous state of the regen process" %
%   N13:3  REGEN_STANDBY_BUFFER  "state The state when the system went to SYSTEM STANDBY" %
%   N13:2  REGEN_ALARM_BUFFER  "STATE The buffered previous state when the system alarm occured" %
%   C5:8  REGEN_PURGE_MINUTES  "COUNTER Regen THe number of minutes the purge step runs" %
% Rung: 32 %
% TITLE: REGEN COOL WALL %
% SYSTEM ALARM
% If the state of this machine is REGEN COOL WALL and the state of the system is SYSTEM ALARM, then buffer the state of this machine and go to the REGEN STANDBY state %
SOR EQU N13:0 N9:35 EQU N10:0 N9:3 BST MOV N9:35 N13:2 NXB MOV N9:29 N13:0 BND EOR
%   N13:0  REGEN_STATE  "<datalog> STATE The current state of the regen process" %
%   N9:35  REGEN_COOL_WALL  "STATE Regen Cool wall" %
%   N10:0  SYSTEM_STATE  "<datalog> STATE The current state of the system" %
%   N9:3  SYSTEM_ALARM  "STATE System Alarm" %
%   N13:2  REGEN_ALARM_BUFFER  "STATE The buffered previous state when the system alarm occured" %
%   N9:29  REGEN_IDLE  "STATE Regen Idle" %
% Rung: 33 %
% REGEN ALARM
% If the state of this machine is REGEN STANDBY and a Regen Alarm occurs, go to the REGEN ALARM state %
SOR EQU N13:0 N9:35 EQU N10:0 N9:1 XIC B34:2/0 BST MOV N9:35 N13:1 NXB MOV N9:37 N13:0 BND EOR
%   N13:0  REGEN_STATE  "<datalog> STATE The current state of the regen process" %
%   N9:35  REGEN_COOL_WALL  "STATE Regen Cool wall" %
%   N10:0  SYSTEM_STATE  "<datalog> STATE The current state of the system" %
%   N9:1  SYSTEM_PROCESS  "STATE System Process" %
%   B34:2/0  REGEN_ALARM_FLAG %
%   N13:1  REGEN_BUFFER  "STATE The buffered, previous state of the regen process" %
%   N9:37  REGEN_ALARM  "STATE Regen Alarm" %

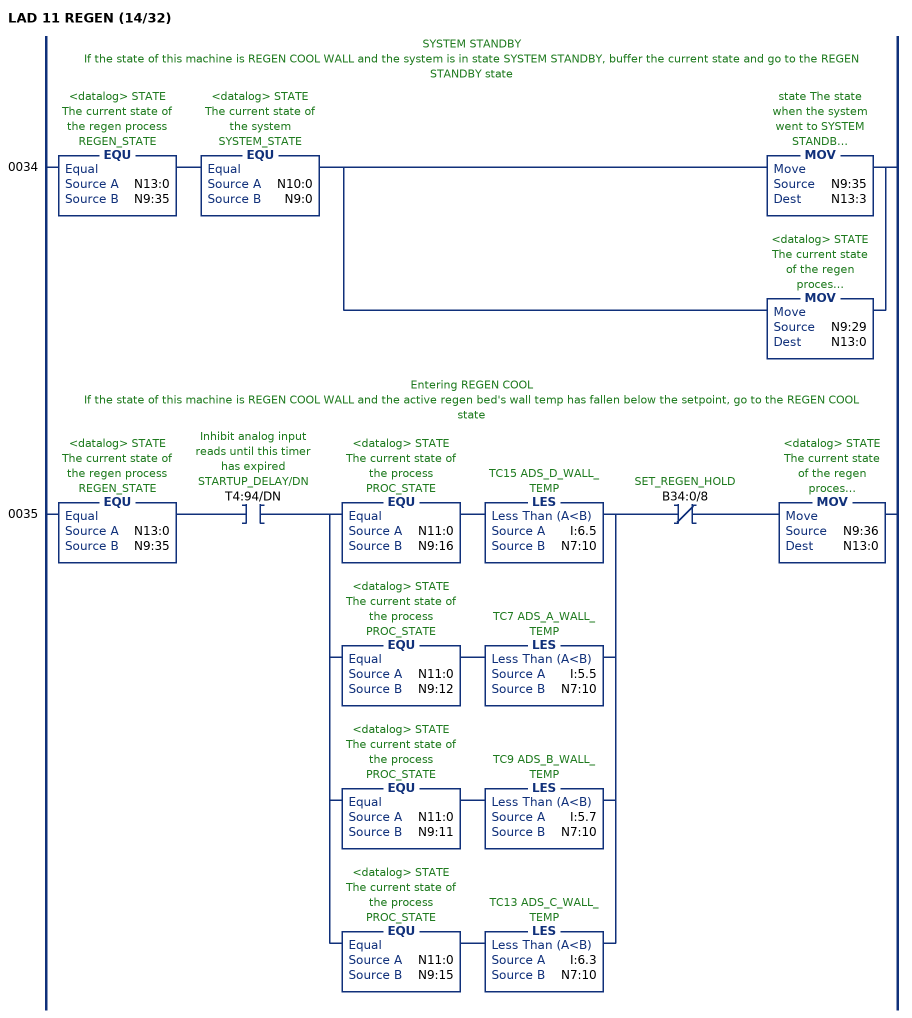
% Rung: 34 %
% SYSTEM STANDBY
% If the state of this machine is REGEN COOL WALL and the system is in state SYSTEM STANDBY, buffer the current state and go to the REGEN STANDBY state %
SOR EQU N13:0 N9:35 EQU N10:0 N9:0 BST MOV N9:35 N13:3 NXB MOV N9:29 N13:0 BND EOR
%   N13:0  REGEN_STATE  "<datalog> STATE The current state of the regen process" %
%   N9:35  REGEN_COOL_WALL  "STATE Regen Cool wall" %
%   N10:0  SYSTEM_STATE  "<datalog> STATE The current state of the system" %
%   N9:0  SYSTEM_STANDBY  "STATE System Standby" %
%   N13:3  REGEN_STANDBY_BUFFER  "state The state when the system went to SYSTEM STANDBY" %
%   N9:29  REGEN_IDLE  "STATE Regen Idle" %
% Rung: 35 %
% Entering REGEN COOL
% If the state of this machine is REGEN COOL WALL and the active regen bed's wall temp has fallen below the setpoint, go to the REGEN COOL state %
SOR EQU N13:0 N9:35 XIC T4:94/DN BST EQU N11:0 N9:16 LES I:6.5 N7:10 NXB EQU N11:0 N9:12 LES I:5.5 N7:10 NXB EQU N11:0 N9:11 LES I:5.7 N7:10 NXB EQU N11:0 N9:15 LES I:6.3 N7:10 BND XIO B34:0/8 MOV N9:36 N13:0 EOR
%   N13:0  REGEN_STATE  "<datalog> STATE The current state of the regen process" %
%   N9:35  REGEN_COOL_WALL  "STATE Regen Cool wall" %
%   T4:94  STARTUP_DELAY  "Inhibit analog input reads until this timer has expired" %
%   N11:0  PROC_STATE  "<datalog> STATE The current state of the process" %
%   N9:16  PROC_REGEN_D  "STATE Process Regen D" %
%   I:6.5  ADS_D_WALL_TEMP  "TC15" %
%   N7:10  ADS_WALL_TEMP_COOL  "CONFIG The temp at which the adsorber wall is deemed to be cool enough to purify" %
%   N9:12  PROC_REGEN_A  "STATE Process Regen A" %
%   I:5.5  ADS_A_WALL_TEMP  "TC7" %
%   N9:11  PROC_REGEN_B  "STATE Process Regen B" %
%   I:5.7  ADS_B_WALL_TEMP  "TC9" %
%   N9:15  PROC_REGEN_C  "STATE Process Regen C" %
%   I:6.3  ADS_C_WALL_TEMP  "TC13" %
%   B34:0/8  SET_REGEN_HOLD %
%   N9:36  REGEN_COOL  "STATE Regen Cool" %

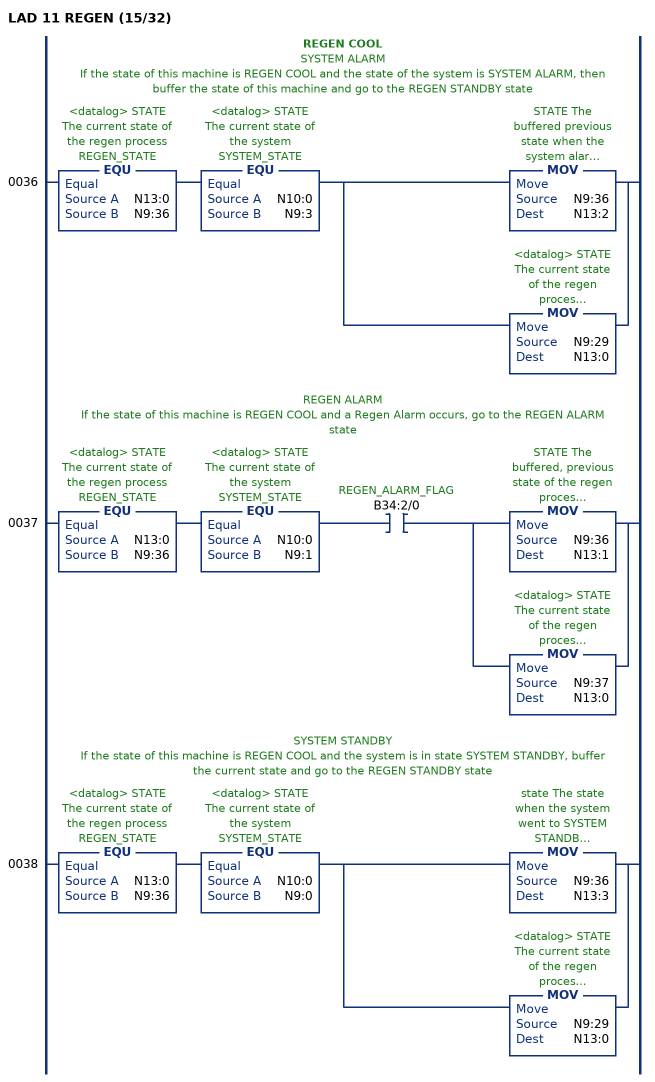
% Rung: 36 %
% TITLE: REGEN COOL %
% SYSTEM ALARM
% If the state of this machine is REGEN COOL and the state of the system is SYSTEM ALARM, then buffer the state of this machine and go to the REGEN STANDBY state %
SOR EQU N13:0 N9:36 EQU N10:0 N9:3 BST MOV N9:36 N13:2 NXB MOV N9:29 N13:0 BND EOR
%   N13:0  REGEN_STATE  "<datalog> STATE The current state of the regen process" %
%   N9:36  REGEN_COOL  "STATE Regen Cool" %
%   N10:0  SYSTEM_STATE  "<datalog> STATE The current state of the system" %
%   N9:3  SYSTEM_ALARM  "STATE System Alarm" %
%   N13:2  REGEN_ALARM_BUFFER  "STATE The buffered previous state when the system alarm occured" %
%   N9:29  REGEN_IDLE  "STATE Regen Idle" %
% Rung: 37 %
% REGEN ALARM
% If the state of this machine is REGEN COOL and a Regen Alarm occurs, go to the REGEN ALARM state %
SOR EQU N13:0 N9:36 EQU N10:0 N9:1 XIC B34:2/0 BST MOV N9:36 N13:1 NXB MOV N9:37 N13:0 BND EOR
%   N13:0  REGEN_STATE  "<datalog> STATE The current state of the regen process" %
%   N9:36  REGEN_COOL  "STATE Regen Cool" %
%   N10:0  SYSTEM_STATE  "<datalog> STATE The current state of the system" %
%   N9:1  SYSTEM_PROCESS  "STATE System Process" %
%   B34:2/0  REGEN_ALARM_FLAG %
%   N13:1  REGEN_BUFFER  "STATE The buffered, previous state of the regen process" %
%   N9:37  REGEN_ALARM  "STATE Regen Alarm" %
% Rung: 38 %
% SYSTEM STANDBY
% If the state of this machine is REGEN COOL and the system is in state SYSTEM STANDBY, buffer the current state and go to the REGEN STANDBY state %
SOR EQU N13:0 N9:36 EQU N10:0 N9:0 BST MOV N9:36 N13:3 NXB MOV N9:29 N13:0 BND EOR
%   N13:0  REGEN_STATE  "<datalog> STATE The current state of the regen process" %
%   N9:36  REGEN_COOL  "STATE Regen Cool" %
%   N10:0  SYSTEM_STATE  "<datalog> STATE The current state of the system" %
%   N9:0  SYSTEM_STANDBY  "STATE System Standby" %
%   N13:3  REGEN_STANDBY_BUFFER  "state The state when the system went to SYSTEM STANDBY" %
%   N9:29  REGEN_IDLE  "STATE Regen Idle" %

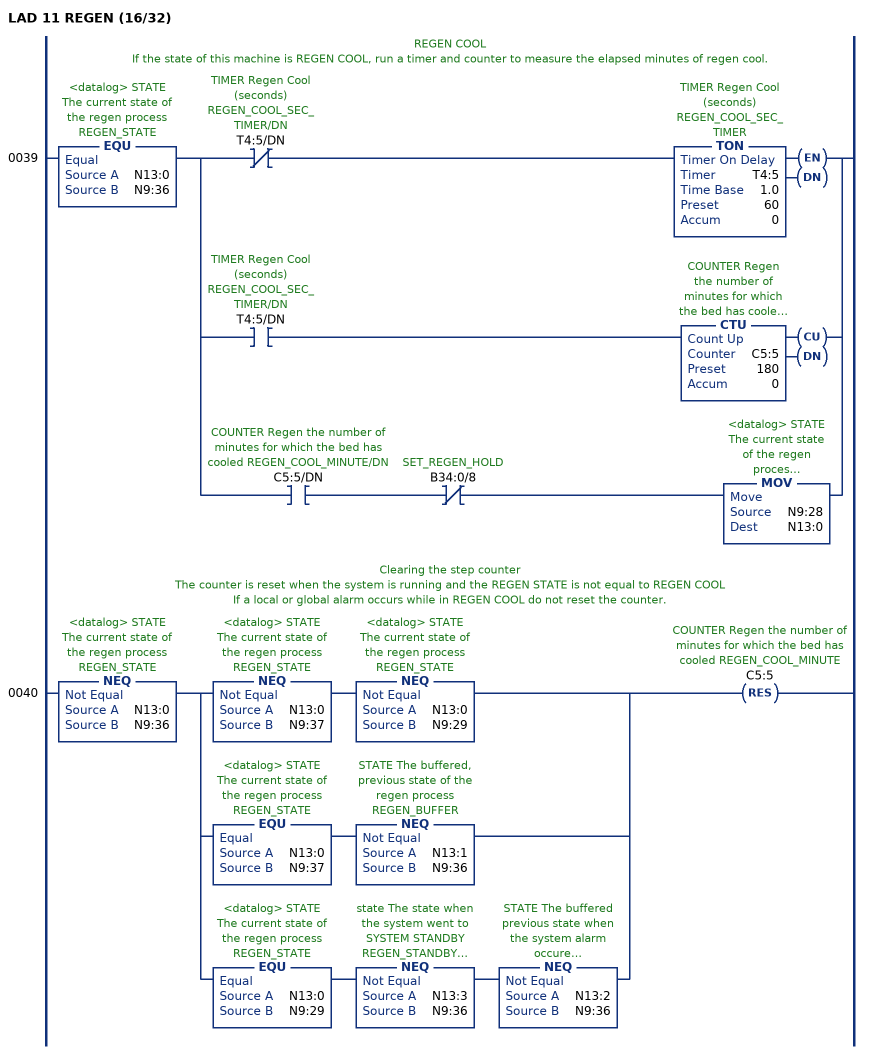
% Rung: 39 %
% REGEN COOL
% If the state of this machine is REGEN COOL, run a timer and counter to measure the elapsed minutes of regen cool. %
SOR EQU N13:0 N9:36 BST XIO T4:5/DN TON T4:5 1.0 60 0 NXB XIC T4:5/DN CTU C5:5 180 0 NXB XIC C5:5/DN XIO B34:0/8 MOV N9:28 N13:0 BND EOR
%   N13:0  REGEN_STATE  "<datalog> STATE The current state of the regen process" %
%   N9:36  REGEN_COOL  "STATE Regen Cool" %
%   T4:5  REGEN_COOL_SEC_TIMER  "TIMER Regen Cool (seconds)" %
%   C5:5  REGEN_COOL_MINUTE  "COUNTER Regen the number of minutes for which the bed has cooled" %
%   B34:0/8  SET_REGEN_HOLD %
%   N9:28  REGEN_VENT_2 %
% Rung: 40 %
% Clearing the step counter
% The counter is reset when the system is running and the REGEN STATE is not equal to REGEN COOL
% If a local or global alarm occurs while in REGEN COOL do not reset the counter. %
SOR NEQ N13:0 N9:36 BST NEQ N13:0 N9:37 NEQ N13:0 N9:29 NXB EQU N13:0 N9:37 NEQ N13:1 N9:36 NXB EQU N13:0 N9:29 NEQ N13:3 N9:36 NEQ N13:2 N9:36 BND RES C5:5 EOR
%   N13:0  REGEN_STATE  "<datalog> STATE The current state of the regen process" %
%   N9:36  REGEN_COOL  "STATE Regen Cool" %
%   N9:37  REGEN_ALARM  "STATE Regen Alarm" %
%   N9:29  REGEN_IDLE  "STATE Regen Idle" %
%   N13:1  REGEN_BUFFER  "STATE The buffered, previous state of the regen process" %
%   N13:3  REGEN_STANDBY_BUFFER  "state The state when the system went to SYSTEM STANDBY" %
%   N13:2  REGEN_ALARM_BUFFER  "STATE The buffered previous state when the system alarm occured" %
%   C5:5  REGEN_COOL_MINUTE  "COUNTER Regen the number of minutes for which the bed has cooled" %

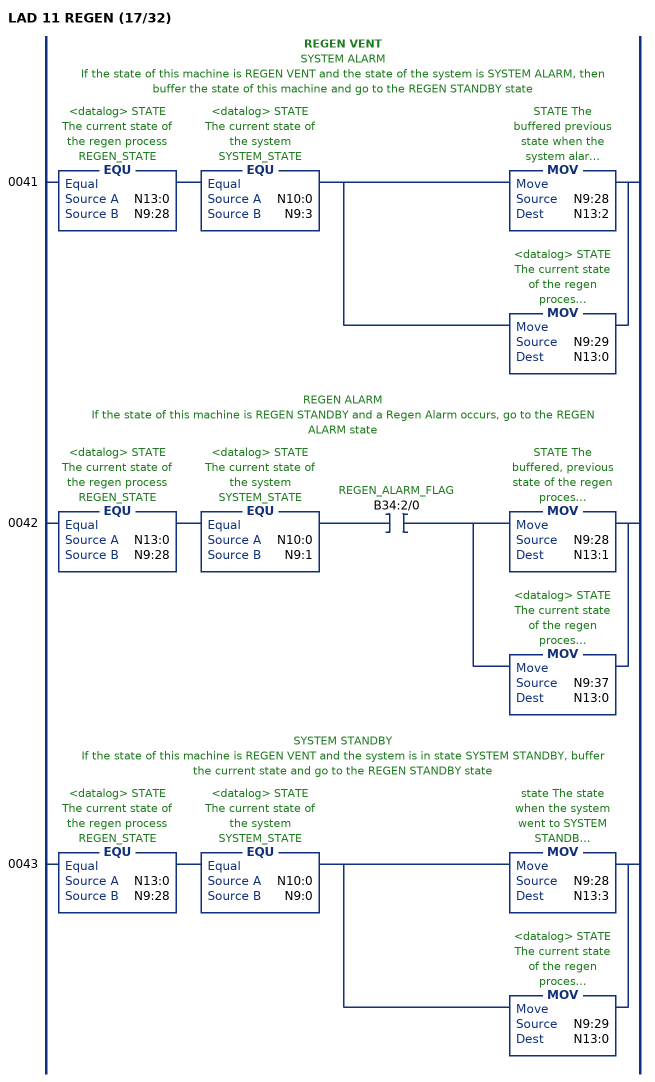
% Rung: 41 %
% TITLE: REGEN VENT %
% SYSTEM ALARM
% If the state of this machine is REGEN VENT and the state of the system is SYSTEM ALARM, then buffer the state of this machine and go to the REGEN STANDBY state %
SOR EQU N13:0 N9:28 EQU N10:0 N9:3 BST MOV N9:28 N13:2 NXB MOV N9:29 N13:0 BND EOR
%   N13:0  REGEN_STATE  "<datalog> STATE The current state of the regen process" %
%   N9:28  REGEN_VENT_2 %
%   N10:0  SYSTEM_STATE  "<datalog> STATE The current state of the system" %
%   N9:3  SYSTEM_ALARM  "STATE System Alarm" %
%   N13:2  REGEN_ALARM_BUFFER  "STATE The buffered previous state when the system alarm occured" %
%   N9:29  REGEN_IDLE  "STATE Regen Idle" %
% Rung: 42 %
% REGEN ALARM
% If the state of this machine is REGEN STANDBY and a Regen Alarm occurs, go to the REGEN ALARM state %
SOR EQU N13:0 N9:28 EQU N10:0 N9:1 XIC B34:2/0 BST MOV N9:28 N13:1 NXB MOV N9:37 N13:0 BND EOR
%   N13:0  REGEN_STATE  "<datalog> STATE The current state of the regen process" %
%   N9:28  REGEN_VENT_2 %
%   N10:0  SYSTEM_STATE  "<datalog> STATE The current state of the system" %
%   N9:1  SYSTEM_PROCESS  "STATE System Process" %
%   B34:2/0  REGEN_ALARM_FLAG %
%   N13:1  REGEN_BUFFER  "STATE The buffered, previous state of the regen process" %
%   N9:37  REGEN_ALARM  "STATE Regen Alarm" %
% Rung: 43 %
% SYSTEM STANDBY
% If the state of this machine is REGEN VENT and the system is in state SYSTEM STANDBY, buffer the current state and go to the REGEN STANDBY state %
SOR EQU N13:0 N9:28 EQU N10:0 N9:0 BST MOV N9:28 N13:3 NXB MOV N9:29 N13:0 BND EOR
%   N13:0  REGEN_STATE  "<datalog> STATE The current state of the regen process" %
%   N9:28  REGEN_VENT_2 %
%   N10:0  SYSTEM_STATE  "<datalog> STATE The current state of the system" %
%   N9:0  SYSTEM_STANDBY  "STATE System Standby" %
%   N13:3  REGEN_STANDBY_BUFFER  "state The state when the system went to SYSTEM STANDBY" %
%   N9:29  REGEN_IDLE  "STATE Regen Idle" %

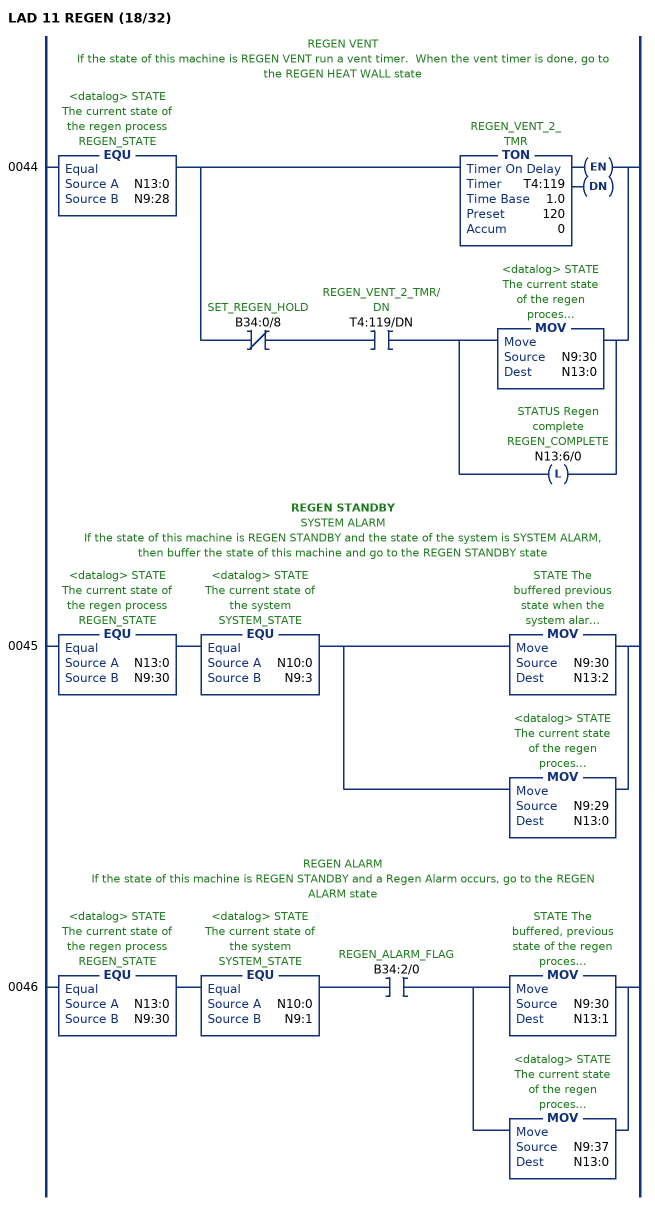
% Rung: 44 %
% REGEN VENT
% If the state of this machine is REGEN VENT run a vent timer.  When the vent timer is done, go to the REGEN HEAT WALL state %
SOR EQU N13:0 N9:28 BST TON T4:119 1.0 120 0 NXB XIO B34:0/8 XIC T4:119/DN BST MOV N9:30 N13:0 NXB OTL N13:6/0 BND BND EOR
%   N13:0  REGEN_STATE  "<datalog> STATE The current state of the regen process" %
%   N9:28  REGEN_VENT_2 %
%   T4:119  REGEN_VENT_2_TMR %
%   B34:0/8  SET_REGEN_HOLD %
%   N9:30  REGEN_STANDBY  "STATE Regen Standby" %
%   N13:6/0  REGEN_COMPLETE  "STATUS Regen complete" %
% Rung: 45 %
% TITLE: REGEN STANDBY %
% SYSTEM ALARM
% If the state of this machine is REGEN STANDBY and the state of the system is SYSTEM ALARM, then buffer the state of this machine and go to the REGEN STANDBY state %
SOR EQU N13:0 N9:30 EQU N10:0 N9:3 BST MOV N9:30 N13:2 NXB MOV N9:29 N13:0 BND EOR
%   N13:0  REGEN_STATE  "<datalog> STATE The current state of the regen process" %
%   N9:30  REGEN_STANDBY  "STATE Regen Standby" %
%   N10:0  SYSTEM_STATE  "<datalog> STATE The current state of the system" %
%   N9:3  SYSTEM_ALARM  "STATE System Alarm" %
%   N13:2  REGEN_ALARM_BUFFER  "STATE The buffered previous state when the system alarm occured" %
%   N9:29  REGEN_IDLE  "STATE Regen Idle" %
% Rung: 46 %
% REGEN ALARM
% If the state of this machine is REGEN STANDBY and a Regen Alarm occurs, go to the REGEN ALARM state %
SOR EQU N13:0 N9:30 EQU N10:0 N9:1 XIC B34:2/0 BST MOV N9:30 N13:1 NXB MOV N9:37 N13:0 BND EOR
%   N13:0  REGEN_STATE  "<datalog> STATE The current state of the regen process" %
%   N9:30  REGEN_STANDBY  "STATE Regen Standby" %
%   N10:0  SYSTEM_STATE  "<datalog> STATE The current state of the system" %
%   N9:1  SYSTEM_PROCESS  "STATE System Process" %
%   B34:2/0  REGEN_ALARM_FLAG %
%   N13:1  REGEN_BUFFER  "STATE The buffered, previous state of the regen process" %
%   N9:37  REGEN_ALARM  "STATE Regen Alarm" %

